otg.CurrentAcceleration[0] := 0;
otg.CurrentAcceleration[1] := 0.2;
otg.CurrentAcceleration[2] := 0;

otg.TargetPosition[0] := 1.0;
otg.TargetPosition[1] := -3.0;
otg.TargetPosition[2] := 2.0;

otg.TargetVelocity[0] := 0.0;
otg.TargetVelocity[1] := 0.0;
otg.TargetVelocity[2] := 0.2;

otg.TargetAcceleration[0] := 0.0;
otg.TargetAcceleration[1] := 0.0;
otg.TargetAcceleration[2] := -0.1;

otg.MaxVelocity[0] := 1;
otg.MaxVelocity[1] := 1;
otg.MaxVelocity[2] := 1;

otg.MaxAcceleration[0] := 1;
otg.MaxAcceleration[1] := 1;
otg.MaxAcceleration[2] := 1;

otg.MaxJerk[0] := 1;
otg.MaxJerk[1] := 1;
otg.MaxJerk[2] := 1;

otg(EnableAutoPropagate := FALSE);
result := otg.State;
AssertEquals_LREAL(otg.Duration, 3.6578610221, 1E-6, Message := ''); 

TEST_FINISHED();
END_METHOD

METHOD Test_FirstStateAtTime
VAR_INST
  otg : Struckig.Otg(0.005, 3) := (
  
    Synchronization := SynchronizationType.TimeSync,
    CurrentPosition :=     [ 0.0, -2.0, 0.0 ],
    CurrentVelocity :=     [ 0.0, 0.0, 0.0 ],
    CurrentAcceleration := [ 0.0, 0.0, 0.0 ],
    TargetPosition :=      [ 1.0, -3.0, 2.0 ],
    TargetVelocity :=      [ 0.0, 0.3, 0.0 ],
    TargetAcceleration :=  [ 0.0, 0.0, 0.0 ],
    MaxVelocity :=         [ 1.0, 1.0, 1.0 ],
    MaxAcceleration :=     [ 1.0, 1.0, 1.0 ],
    MaxJerk :=             [ 1.0, 1.0, 1.0 ]
  );
    
END_VAR
VAR
  result : Struckig.TrajectoryState;
  NewPosition, NewVelocity, NewAcceleration, values : ARRAY[0..Struckig.ParameterList.MaxDoFs] OF LREAL;
  positionExtrema : Struckig.PositionExtremaDesc;
  rtime, rvel, racc : LREAL;
END_VAR
TEST('FirstStateAtTime');

otg();

AssertTrue( otg._profiles[0].firstStateAtPosition(0.0, 0.0, rtime, rvel, racc), message:='' );
AssertEquals_LREAL(0.0, rtime, 1E-9, message:='');

AssertTrue( otg._profiles[0].firstStateAtPosition(0.5, 0.0, rtime, rvel, racc), message:='' );
AssertEquals_LREAL(2.0, rtime, 1E-9, message:='');

AssertTrue( otg._profiles[0].firstStateAtPosition(1.0, 0.0, rtime, rvel, racc), message:='' );
AssertEquals_LREAL(3.9999857615998957, rtime, 1E-9, message:=''); // doctest::Approx(4.0) 

AssertTrue( otg._profiles[1].firstStateAtPosition(-3.0, 0.0, rtime, rvel, racc), message:='' );
AssertEquals_LREAL(2.6004877902, rtime, 1E-9, message:='');

AssertTrue( otg._profiles[1].firstStateAtPosition(-3.1, 0.0, rtime, rvel, racc), message:='' );
AssertEquals_LREAL(2.8644154489, rtime, 1E-9, message:='');

AssertTrue( otg._profiles[2].firstStateAtPosition(0.05, 0.0, rtime, rvel, racc), message:='' );
AssertEquals_LREAL(0.6694329501, rtime, 1E-9, message:='');

AssertFalse( otg._profiles[0].firstStateAtPosition(-1.0, 0.0, rtime, rvel, racc), message:='' );
AssertFalse( otg._profiles[1].firstStateAtPosition(-3.4, 0.0, rtime, rvel, racc), message:='' );

// todo: this test doesn't make sense in the port of ruckig, the method is not exposed in the trajectory class yet
// AssertFalse( ruckig._profiles[6].firstStateAtPosition(6, 0.0, rtime, rvel, racc), message:='' );

TEST_FINISHED();
END_METHOD

METHOD Test_IndependentMinDurations
VAR_INST
  otg : Struckig.Otg(0.005, 3) := (
  
    Synchronization := SynchronizationType.None,
    CurrentPosition :=     [ 0.0, -2.0, 0.0 ],
    CurrentVelocity :=     [ 0.0, 0.0, 0.0 ],
    CurrentAcceleration := [ 0.0, 0.0, 0.0 ],
    TargetPosition :=      [ 1.0, -3.0, 2.0 ],
    TargetVelocity :=      [ 0.0, 0.3, 0.0 ],
    TargetAcceleration :=  [ 0.0, 0.0, 0.0 ],
    MaxVelocity :=         [ 1.0, 1.0, 1.0 ],
    MaxAcceleration :=     [ 1.0, 1.0, 1.0 ],
    MaxJerk :=             [ 1.0, 1.0, 1.0 ]
  );
    
END_VAR
VAR
  result : Struckig.TrajectoryState;
  NewPosition, NewVelocity, NewAcceleration, values : ARRAY[0..Struckig.ParameterList.MaxDoFs] OF LREAL;
  positionExtrema : Struckig.PositionExtremaDesc;
  rtime, rvel, racc : LREAL;
END_VAR
TEST('IndependentMinDurations');

otg();

AssertEquals_LREAL(otg._independentMinDurations[0], 3.1748021039, 1E-9, message:='');
AssertEquals_LREAL(otg._independentMinDurations[1], 3.6860977315, 1E-9, message:='');
AssertEquals_LREAL(otg._independentMinDurations[2], otg.Duration, 1E-9, message:='');

TEST_FINISHED();
END_METHOD

METHOD Test_InvalidInput
VAR_INST
  otg : Struckig.Otg(0.005, 3) := (
  
    Synchronization := SynchronizationType.None,
    CurrentPosition :=     [ 0.0, -2.0, 0.0 ],
    CurrentVelocity :=     [ 0.0, 0.0, 0.0 ],
    CurrentAcceleration := [ 0.0, 0.0, 0.0 ],
    TargetPosition :=      [ 1.0, -3.0, 2.0 ],
    TargetVelocity :=      [ 0.0, 0.3, 0.0 ],
    TargetAcceleration :=  [ 0.0, 0.0, 0.0 ],
    MaxVelocity :=         [ 1.0, 1.0, 1.0 ],
    MaxAcceleration :=     [ 1.0, 1.0, 1.0 ],
    MaxJerk :=             [ 1.0, 1.0, 1.0 ]
  );
    
END_VAR
VAR
  result : Struckig.TrajectoryState;
  NewPosition, NewVelocity, NewAcceleration, values : ARRAY[0..Struckig.ParameterList.MaxDoFs] OF LREAL;
  positionExtrema : Struckig.PositionExtremaDesc;
  rtime, rvel, racc : LREAL;
END_VAR
TEST('InvalidInput');

otg();

otg.TargetVelocity[0] := 2.0;
otg.TargetVelocity[1] := 0.3;
otg.TargetVelocity[2] := 0.0;

otg();

AssertEquals_INT(otg.State, Struckig.TrajectoryState.error, message:='State should be error');
AssertFalse(otg.NewCalculation, message:='ruckig.NewCalculation should be false');

otg.TargetVelocity[0] := 0.2;
otg.TargetVelocity[1] := -0.3;
otg.TargetVelocity[2] := 0.8;

otg();

AssertEquals_INT(otg.State, Struckig.TrajectoryState.busy, message:='State should be busy');
AssertTrue(otg.NewCalculation, message:='ruckig.NewCalculation should be true');

TEST_FINISHED();
END_METHOD

METHOD Test_PerDofSettings
VAR_INST
  otg : Struckig.Otg(0.005, 3) := (
    CurrentPosition :=     [ 0.0, -2.0, 0.0 ],
    CurrentVelocity :=     [ 0.0, 0.0, 0.0 ],
    CurrentAcceleration := [ 0.0, 0.0, 0.0 ],
    TargetPosition :=      [ 1.0, -3.0, 2.0 ],
    TargetVelocity :=      [ 0.0, 0.3, 0.0 ],
    TargetAcceleration :=  [ 0.0, 0.0, 0.0 ],
    MaxVelocity :=         [ 1.0, 1.0, 1.0 ],
    MaxAcceleration :=     [ 1.0, 1.0, 1.0 ],
    MaxJerk :=             [ 1.0, 1.0, 1.0 ]
  );
    
END_VAR
VAR
  result : Struckig.TrajectoryState;
  NewPosition, NewVelocity, NewAcceleration, values : ARRAY[0..Struckig.ParameterList.MaxDoFs] OF LREAL;
  NewSection : INT;
  positionExtrema : Struckig.PositionExtremaDesc;
  rtime, rvel, racc : LREAL;
END_VAR
TEST('PerDofSettings');

otg();
AssertEquals_INT(otg.State, Struckig.TrajectoryState.Busy, message:='State should be busy');
AssertEquals_LREAL(otg.Duration, 4, 1E-6, message:='Duration not met');

otg.AtTime(2.0, ADR(NewPosition), ADR(NewVelocity), ADR(NewAcceleration), ADR(NewSection));
values[0] := 0.5;
values[1] := -2.6871268303;
values[2] :=  1.0;
AssertArrayEquals_LREAL(values, NewPosition, 1E-6, message:='Position not met');


otg.ControlInterface := ControlInterfaceType.Velocity;
otg();
AssertEquals_INT(otg.State, Struckig.TrajectoryState.Busy, message:='State should be busy');
AssertEquals_LREAL(otg.Duration, 1.095445115, 1E-6, message:='Duration not met');

otg.AtTime(1.0, ADR(NewPosition), ADR(NewVelocity), ADR(NewAcceleration), ADR(NewSection));
values[0] := 0.0;
values[1] := -1.8641718534;
values[2] :=  0.0;
AssertArrayEquals_LREAL(values, NewPosition, 1E-6, message:='Position not met');


otg.PerDofControlInterface[0] := ControlInterfaceType.Position;
otg.PerDofControlInterface[1] := ControlInterfaceType.Velocity;
otg.PerDofControlInterface[2] := ControlInterfaceType.Position;
otg();
AssertEquals_INT(otg.State, Struckig.TrajectoryState.Busy, message:='State should be busy');
AssertEquals_LREAL(otg.Duration, 4.0, 1E-6, message:='Duration not met');

otg.AtTime(2.0, ADR(NewPosition), ADR(NewVelocity), ADR(NewAcceleration), ADR(NewSection));
values[0] := 0.5;
values[1] := -1.8528486838;
values[2] := 1.0;
AssertArrayEquals_LREAL(values, NewPosition, 1E-6, message:='Position not met');


otg.PerDofSynchronization[0] := SynchronizationType.TimeSync;
otg.PerDofSynchronization[1] := SynchronizationType.None;
otg.PerDofSynchronization[2] := SynchronizationType.TimeSync;
otg();
AssertEquals_INT(otg.State, Struckig.TrajectoryState.Busy, message:='State should be busy');
AssertEquals_LREAL(otg.Duration, 4.0, 1E-6, message:='Duration not met');

otg.AtTime(2.0, ADR(NewPosition), ADR(NewVelocity), ADR(NewAcceleration), ADR(NewSection));
values[0] := 0.5;
values[1] := -1.5643167673;
values[2] := 1.0;
AssertArrayEquals_LREAL(values, NewPosition, 1E-6, message:='Position not met');

otg.ControlInterface := ControlInterfaceType.Position;
otg.PerDofControlInterface[0] := ControlInterfaceType.Undefined;
otg.PerDofControlInterface[1] := ControlInterfaceType.Undefined;
otg.PerDofControlInterface[2] := ControlInterfaceType.Undefined;
otg.PerDofSynchronization[0] := SynchronizationType.None;
otg.PerDofSynchronization[1] := SynchronizationType.TimeSync;
otg.PerDofSynchronization[2] := SynchronizationType.TimeSync;
otg();
AssertEquals_INT(otg.State, Struckig.TrajectoryState.Busy, message:='State should be busy');
AssertEquals_LREAL(otg.Duration, 4.0, 1E-6, message:='Duration not met');

otg.AtTime(2.0, ADR(NewPosition), ADR(NewVelocity), ADR(NewAcceleration), ADR(NewSection));
values[0] := 0.7482143874;
values[1] := -2.6871268303;
values[2] := 1.0;
AssertArrayEquals_LREAL(values, NewPosition, 1E-6, message:='Position not met');

TEST_FINISHED();
END_METHOD

METHOD Test_PerDofSettings_1
VAR_INST
  otg : Struckig.Otg(0.005, 3) := (
    CurrentPosition :=     [ 0.0, 0.0, 0.0 ],
    CurrentVelocity :=     [ 0.0, 0.0, 0.0 ],
    CurrentAcceleration := [ 0.0, 0.0, 0.0 ],
    TargetPosition :=      [ 35, 35, 35 ],
    TargetVelocity :=      [ 125, 125, 100 ],
    TargetAcceleration :=  [ 0.0, 0.0, 0.0 ],
    MaxVelocity :=         [ 125, 125, 100 ],
    MaxAcceleration :=     [ 2000, 2000, 2000 ],
    MaxJerk :=             [ 20000, 20000, 20000 ]
  );
    
END_VAR
VAR
  result : Struckig.TrajectoryState;
END_VAR
TEST('PerDofSettings_1');

otg.ControlInterface := ControlInterfaceType.Position;
otg.PerDofControlInterface[0] := ControlInterfaceType.Undefined;
otg.PerDofControlInterface[1] := ControlInterfaceType.Undefined;
otg.PerDofControlInterface[2] := ControlInterfaceType.Undefined;
otg.PerDofSynchronization[0] := SynchronizationType.TimeSync;
otg.PerDofSynchronization[1] := SynchronizationType.TimeSync;
otg.PerDofSynchronization[2] := SynchronizationType.None;
otg();
AssertEquals_INT(otg.State, Struckig.TrajectoryState.Busy, message:='State should be busy');
AssertEquals_LREAL(otg.Duration, 0.4207106781, 1E-6, message:='Duration not met');


otg.CurrentPosition[0] := 0;
otg.CurrentPosition[1] := -2;
otg.CurrentPosition[2] := 0;

otg.CurrentVelocity[0] := 0;
otg.CurrentVelocity[1] := 0.2;
otg.CurrentVelocity[2] := 0;

otg.CurrentAcceleration[0] := 0;
otg.CurrentAcceleration[1] := 0.2;
otg.CurrentAcceleration[2] := 0;

otg.TargetPosition[0] := 1.0;
otg.TargetPosition[1] := -3.0;
otg.TargetPosition[2] := 2.0;

otg.TargetVelocity[0] := 0.0;
otg.TargetVelocity[1] := 0.0;
otg.TargetVelocity[2] := 0.2;

otg.TargetAcceleration[0] := 0.0;
otg.TargetAcceleration[1] := 0.0;
otg.TargetAcceleration[2] := -0.1;

otg.MaxVelocity[0] := 1;
otg.MaxVelocity[1] := 1;
otg.MaxVelocity[2] := 1;

otg.MaxAcceleration[0] := 1;
otg.MaxAcceleration[1] := 1;
otg.MaxAcceleration[2] := 1;

otg.MaxJerk[0] := 1;
otg.MaxJerk[1] := 1;
otg.MaxJerk[2] := 1;

otg.PerDofSynchronization[0] := SynchronizationType.None;
otg.PerDofSynchronization[1] := SynchronizationType.None;
otg.PerDofSynchronization[2] := SynchronizationType.TimeSync;

otg();
AssertEquals_INT(otg.State, Struckig.TrajectoryState.Busy, message:='State should be busy');
AssertEquals_LREAL(otg.Duration, 3.7885667284, 1E-6, message:='Duration not met');

otg.PerDofSynchronization[0] := SynchronizationType.None;
otg.PerDofSynchronization[1] := SynchronizationType.TimeSync;
otg.PerDofSynchronization[2] := SynchronizationType.None;

otg();
AssertEquals_INT(otg.State, Struckig.TrajectoryState.Busy, message:='State should be busy');
AssertEquals_LREAL(otg.Duration, 3.7885667284, 1E-6, message:='Duration not met');

otg.Enabled[0] := TRUE;
otg.Enabled[1] := FALSE;
otg.Enabled[2] := TRUE;

otg();
AssertEquals_INT(otg.State, Struckig.TrajectoryState.Busy, message:='State should be busy');
AssertEquals_LREAL(otg.Duration, 3.6578610221, 1E-6, message:='Duration not met');

TEST_FINISHED();
END_METHOD

METHOD Test_PhaseSynchronization
VAR_INST
  otg : Struckig.Otg(0.005, 3) := (
    Synchronization := SynchronizationType.Phase,
    CurrentPosition :=     [ 0.0, -2.0, 0.0 ],
    TargetPosition :=      [ 1.0, -3.0, 2.0 ],
    MaxVelocity :=         [ 1.0, 1.0, 1.0 ],
    MaxAcceleration :=     [ 1.0, 1.0, 1.0 ],
    MaxJerk :=             [ 1.0, 1.0, 1.0 ]
  ); 
END_VAR
VAR
  result : Struckig.TrajectoryState;
  busy : Struckig.TrajectoryState := Struckig.TrajectoryState.Busy;
  NewSection : INT;
  NewPosition, NewVelocity, NewAcceleration, values : ARRAY[0..Struckig.ParameterList.MaxDoFs] OF LREAL;
  positionExtrema : Struckig.PositionExtremaDesc;
  rtime, rvel, racc : LREAL;
END_VAR
TEST('PhaseSynchronization');

otg();
result := otg.State;
AssertEquals(busy, result, Message := '');
AssertEquals_LREAL(otg.Duration, 4.0, 1E-6, Message := ''); 
otg.AtTime(1.0, ADR(NewPosition), ADR(NewVelocity), ADR(NewAcceleration), ADR(NewSection));
values[0] := 0.0833333333;
values[1] := -2.0833333333;
values[2] := 0.1666666667;
AssertArrayEquals_LREAL(values, NewPosition, 1E-6, '');




otg.CurrentPosition[0] := 0.0;
otg.CurrentPosition[1] := -2.0;
otg.CurrentPosition[2] := 0.0;

otg.TargetPosition[0] := 10.0;
otg.TargetPosition[1] := -3.0;
otg.TargetPosition[2] := 2.0;

otg.MaxVelocity[0] := 10.0;
otg.MaxVelocity[1] := 2.0;
otg.MaxVelocity[2] := 1.0;

otg.MaxAcceleration[0] := 10.0;
otg.MaxAcceleration[1] := 2.0;
otg.MaxAcceleration[2] := 1.0;

otg.MaxJerk[0] := 10.0;
otg.MaxJerk[1] := 2.0;
otg.MaxJerk[2] := 1.0;

otg();
result := otg.State;
AssertEquals(busy, result, Message := '');
AssertEquals_LREAL(otg.Duration, 4.0, 1E-6, Message := ''); 
otg.AtTime(1.0, ADR(NewPosition), ADR(NewVelocity), ADR(NewAcceleration), ADR(NewSection));
values[0] := 0.8333333333;
values[1] := -2.0833333333;
values[2] := 0.1666666667;
AssertArrayEquals_LREAL(values, NewPosition, 1E-6, '');

TEST_FINISHED();
END_METHOD

METHOD Test_PositionExtrema
VAR_INST
  otg : Struckig.Otg(0.005, 3) := (
    Synchronization := SynchronizationType.TimeSync,
    CurrentPosition :=     [ 0.0, -2.0, 0.0 ],
    TargetPosition :=      [ 1.0, -3.0, 2.0 ],
    TargetVelocity :=      [ 0.0, 0.3, 0.0 ],
    MaxVelocity :=         [ 1.0, 1.0, 1.0 ],
    MaxAcceleration :=     [ 1.0, 1.0, 1.0 ],
    MaxJerk :=             [ 1.0, 1.0, 1.0 ]
  );     
END_VAR
VAR
  result : Struckig.TrajectoryState;
  NewPosition, NewVelocity, NewAcceleration, values : ARRAY[0..Struckig.ParameterList.MaxDoFs] OF LREAL;
  positionExtrema : Struckig.PositionExtremaDesc;
  rtime, rvel, racc : LREAL;
END_VAR
TEST('PositionExtrema');

otg();

positionExtrema := otg._profiles[0].positionExtrema();
AssertEquals_LREAL(4.0, positionExtrema.Tmax, 1E-9, message:='Profile[0] Tmax incorrect');
AssertEquals_LREAL(1.0, positionExtrema.Maximum, 1E-9, message:='Profile[0] maximum incorrect');
AssertEquals_LREAL(0.0, positionExtrema.Tmin, 1E-9, message:='Profile[0] Tmin incorrect');
AssertEquals_LREAL(0.0, positionExtrema.Minimum, 1E-9, message:='Profile[0] minimum incorrect');

positionExtrema := otg._profiles[1].positionExtrema();
AssertEquals_LREAL(0.0, positionExtrema.Tmax, 1E-9, message:='Profile[1] Tmax incorrect');
AssertEquals_LREAL(-2.0, positionExtrema.Maximum, 1E-9, message:='Profile[1] maximum incorrect');
AssertEquals_LREAL(3.2254033308, positionExtrema.Tmin, 1E-9, message:='Profile[1] Tmin incorrect');
AssertEquals_LREAL(-3.1549193338, positionExtrema.Minimum, 1E-9, message:='Profile[1] minimum incorrect');

positionExtrema := otg._profiles[2].positionExtrema();
AssertEquals_LREAL(4.0, positionExtrema.Tmax, 1E-9, message:='Profile[2] Tmax incorrect');
AssertEquals_LREAL(2.0, positionExtrema.Maximum, 1E-9, message:='Profile[2] maximum incorrect');
AssertEquals_LREAL(0.0, positionExtrema.Tmin, 1E-9, message:='Profile[2] Tmin incorrect');
AssertEquals_LREAL(0.0, positionExtrema.Minimum, 1E-9, message:='Profile[2] minimum incorrect');

TEST_FINISHED();
END_METHOD

END_FUNCTION_BLOCK

// ---- POUs/DebuggedExamplesTest.TcPOU
FUNCTION_BLOCK DebuggedExamplesTest EXTENDS TcUnit.FB_TestSuite

Test_Trajectory_HasTargetVelocity_HasTargetAcceleration();

METHOD Test_Trajectory_HasTargetVelocity_HasTargetAcceleration
VAR_INST
  ruckig : Struckig.Otg(0.001, 3) := (
  
    Synchronization := SynchronizationType.TimeSync,        
    MaxVelocity := [ 2000.00000000000000000000, 2000.00000000000000000000, 2000.00000000000000000000 ],
    MaxAcceleration := [ 20000.00000000000000000000, 20000.00000000000000000000, 20000.00000000000000000000 ],
    MaxJerk := [ 800000.00000000000000000000, 800000.00000000000000000000, 800000.00000000000000000000 ],
    CurrentPosition := [ -54.94342725690739825950, -71.16344937395382430623, -99.92141940871530891854 ],
    CurrentVelocity := [ 203.04708462957614756306, -87.88615914847480325989, -244.40742200449426491105 ],
    CurrentAcceleration := [ -9414.24830241836389177479, 3433.58972946014000626747, -1048.10905719350193976425 ],
    TargetPosition := [ -30.34627507739200780179, 41.33313071646210801191, 94.47974487226861128875 ],
    TargetVelocity := [ -104.33706621689987059654, -659.36109838358197521302, 811.33117925934993763804 ],
    TargetAcceleration := [ 523.43053514200096287823, 100.75104632855459385610, 320.80199262854853259341 ]
  );
  
  positionExtrema : Struckig.PositionExtremaDesc;
END_VAR
TEST('Trajectory_Profile[1]_Step2_TimeVel');

ruckig();

// Check total duration of profiles
AssertEquals_LREAL(Expected := 0.22338925049474450679, Actual := ruckig.Duration, DELTA := 1E-8, Message := 'Duration incorrect');

// Check duration for each phase
positionExtrema := ruckig._profiles[0].positionExtrema();
AssertEquals_LREAL(0.20657109030979783904, positionExtrema.Tmax, 1E-9, message:='Profile[0] Tmax incorrect');
AssertEquals_LREAL(-29.15176131633907630203, positionExtrema.Maximum, 1E-9, message:='Profile[0] maximum incorrect');
AssertEquals_LREAL(0.00000000000000000000, positionExtrema.Tmin, 1E-9, message:='Profile[0] Tmin incorrect');
AssertEquals_LREAL(-54.94342725690739825950, positionExtrema.Minimum, 1E-9, message:='Profile[0] minimum incorrect');

positionExtrema := ruckig._profiles[1].positionExtrema();
AssertEquals_LREAL(0.19826331168683380968, positionExtrema.Tmax, 1E-9, message:='Profile[1] Tmax incorrect');
AssertEquals_LREAL(55.81702313192161568622, positionExtrema.Maximum, 1E-9, message:='Profile[1] maximum incorrect');
AssertEquals_LREAL(0.01113968648909354625, positionExtrema.Tmin, 1E-9, message:='Profile[1] Tmin incorrect');
AssertEquals_LREAL(-71.74511835894615785492, positionExtrema.Minimum, 1E-9, message:='Profile[1] minimum incorrect');

positionExtrema := ruckig._profiles[2].positionExtrema();
AssertEquals_LREAL(0.22338925049474447904, positionExtrema.Tmax, 1E-9, message:='Profile[2] Tmax incorrect');
AssertEquals_LREAL(94.47974487226861128875, positionExtrema.Maximum, 1E-9, message:='Profile[2] maximum incorrect');
AssertEquals_LREAL(0.02606362117094545780, positionExtrema.Tmin, 1E-9, message:='Profile[2] Tmin incorrect');
AssertEquals_LREAL(-104.28684661857214166503, positionExtrema.Minimum, 1E-9, message:='Profile[2] minimum incorrect');
   

TEST_FINISHED();
END_METHOD

END_FUNCTION_BLOCK

// ---- POUs/TargetPosTest.TcPOU
FUNCTION_BLOCK TargetPosTest EXTENDS TcUnit.FB_TestSuite
VAR
  ruckig : Struckig.Otg(0.001, 3) := (
  
    Synchronization := SynchronizationType.TimeSync,        
    MaxVelocity := [ 2000.00000000000000000000, 2000.00000000000000000000, 2000.00000000000000000000 ],
    MaxAcceleration := [ 20000.00000000000000000000, 20000.00000000000000000000, 20000.00000000000000000000 ],
    MaxJerk := [ 800000.00000000000000000000, 800000.00000000000000000000, 800000.00000000000000000000 ],
    CurrentPosition := [ 48.86656216713086564596, 31.55963588984187140341, -13.09422790776093847853 ],
    CurrentVelocity := [ -274.21841080128081102885, -440.94461360926254656079, -764.75678162210920163488 ],
    CurrentAcceleration := [ -1478.09700836416959646158, 686.79611869591644790489, -9263.72976579731221136171 ],
    TargetPosition := [ 25.57994474955607699940, -15.83091418217283319336, -38.97164514571973370494 ],
    TargetVelocity := [ 0.00000000000000000000, 0.00000000000000000000, 0.00000000000000000000 ],
    TargetAcceleration := [ 0.00000000000000000000, 0.00000000000000000000, 0.00000000000000000000 ]
  );
  
  positionExtrema : Struckig.PositionExtremaDesc;  
END_VAR

Test_Trajectory_2();;
Test_Trajectory_5();
Test_Trajectory_6();
Test_Trajectory_7();
Test_Trajectory_12();
Test_Trajectory_16(); // this test required to do a more precise implementation of cbrt
Test_Trajectory_30();
Test_Trajectory_32();
Test_Trajectory_33();
Test_Trajectory_40();
Test_Trajectory_49();
Test_Trajectory_53();
Test_Trajectory_59();
Test_Trajectory_62();
Test_Trajectory_64();
Test_Trajectory_65();
Test_Trajectory_68();

METHOD Test_Trajectory_12
VAR_INST
  ruckig : Struckig.Otg(0.001, 3) := (
  
    Synchronization := SynchronizationType.TimeSync,        
    MaxVelocity := [ 2000.00000000000000000000, 2000.00000000000000000000, 2000.00000000000000000000 ],
    MaxAcceleration := [ 20000.00000000000000000000, 20000.00000000000000000000, 20000.00000000000000000000 ],
    MaxJerk := [ 800000.00000000000000000000, 800000.00000000000000000000, 800000.00000000000000000000 ],
    CurrentPosition := [ 12.15863849634686744139, 83.56438022017914590833, -29.82534868849941744884 ],
    CurrentVelocity := [ -881.54677264260010360886, -40.22247547933807254594, 795.30816871835008896596 ],
    CurrentAcceleration := [ 6802.73049394882036722265, -2844.95338607063877134351, -3652.21806306270900677191 ],
    TargetPosition := [ 61.24855302996508044089, -54.65891429617437324850, 65.64407005892678625969 ],
    TargetVelocity := [ 0.00000000000000000000, 0.00000000000000000000, 0.00000000000000000000 ],
    TargetAcceleration := [ 0.00000000000000000000, 0.00000000000000000000, 0.00000000000000000000 ]
  );
  
  positionExtrema : Struckig.PositionExtremaDesc;
END_VAR
TEST('Trajectory_12');

ruckig();

// Check total duration of profiles
AssertEquals_LREAL(Expected := 0.18765626933931714437, Actual := ruckig.Duration, DELTA := 1E-8, Message := 'Duration incorrect');

// Check duration for each phase
positionExtrema := ruckig._profiles[0].positionExtrema();
AssertEquals_LREAL(0.18765626933931711662, positionExtrema.Tmax, 1E-9, message:='Profile[0] Tmax incorrect');
AssertEquals_LREAL(61.24855302996508044089, positionExtrema.Maximum, 1E-9, message:='Profile[0] maximum incorrect');
AssertEquals_LREAL(0.01649658688256397387, positionExtrema.Tmin, 1E-9, message:='Profile[0] Tmin incorrect');
AssertEquals_LREAL(-0.85965741863935996037, positionExtrema.Minimum, 1E-9, message:='Profile[0] minimum incorrect');

positionExtrema := ruckig._profiles[1].positionExtrema();
AssertEquals_LREAL(0.00000000000000000000, positionExtrema.Tmax, 1E-9, message:='Profile[1] Tmax incorrect');
AssertEquals_LREAL(83.56438022017914590833, positionExtrema.Maximum, 1E-9, message:='Profile[1] maximum incorrect');
AssertEquals_LREAL(0.18765626933931714437, positionExtrema.Tmin, 1E-9, message:='Profile[1] Tmin incorrect');
AssertEquals_LREAL(-54.65891429617437324850, positionExtrema.Minimum, 1E-9, message:='Profile[1] minimum incorrect');

positionExtrema := ruckig._profiles[2].positionExtrema();
AssertEquals_LREAL(0.18765626933931711662, positionExtrema.Tmax, 1E-9, message:='Profile[2] Tmax incorrect');
AssertEquals_LREAL(65.64407005892678625969, positionExtrema.Maximum, 1E-9, message:='Profile[2] maximum incorrect');
AssertEquals_LREAL(0.00000000000000000000, positionExtrema.Tmin, 1E-9, message:='Profile[2] Tmin incorrect');
AssertEquals_LREAL(-29.82534868849941744884, positionExtrema.Minimum, 1E-9, message:='Profile[2] minimum incorrect');
   

TEST_FINISHED();
END_METHOD

METHOD Test_Trajectory_16
VAR_INST
  ruckig : Struckig.Otg(0.001, 3) := (
  
    Synchronization := SynchronizationType.TimeSync,        
    MaxVelocity := [ 2000.00000000000000000000, 2000.00000000000000000000, 2000.00000000000000000000 ],
    MaxAcceleration := [ 20000.00000000000000000000, 20000.00000000000000000000, 20000.00000000000000000000 ],
    MaxJerk := [ 800000.00000000000000000000, 800000.00000000000000000000, 800000.00000000000000000000 ],
    CurrentPosition := [ 8.21667911707363884943, -42.91905125747626215116, 48.44417367414695263506 ],
    CurrentVelocity := [ -786.82135287550590874162, 724.24582523622666485608, -678.96507198447488917736 ],
    CurrentAcceleration := [ 2775.55640569175011478364, 5006.65330127050037845038, -1991.17849814757664717035 ],
    TargetPosition := [ -91.18523630560480341956, 39.65724384459844031880, 80.00859285567460688071 ],
    TargetVelocity := [ 0.00000000000000000000, 0.00000000000000000000, 0.00000000000000000000 ],
    TargetAcceleration := [ 0.00000000000000000000, 0.00000000000000000000, 0.00000000000000000000 ]
  );
  
  positionExtrema : Struckig.PositionExtremaDesc;
END_VAR
TEST('Trajectory_16');

ruckig();

// Check total duration of profiles
AssertEquals_LREAL(Expected := 0.16787256653000462436, Actual := ruckig.Duration, DELTA := 1E-8, Message := 'Duration incorrect');

// Check duration for each phase
positionExtrema := ruckig._profiles[0].positionExtrema();
AssertEquals_LREAL(0, positionExtrema.Tmax, 1E-9, message:='Profile[0] Tmax incorrect');
AssertEquals_LREAL(8.2166791170736388494, positionExtrema.Maximum, 1E-9, message:='Profile[0] maximum incorrect');
AssertEquals_LREAL(0.16787256653000462436, positionExtrema.Tmin, 1E-9, message:='Profile[0] Tmin incorrect');
AssertEquals_LREAL(-91.18523630560480342, positionExtrema.Minimum, 1E-9, message:='Profile[0] minimum incorrect');

positionExtrema := ruckig._profiles[1].positionExtrema();
AssertEquals_LREAL(0.16787256609842091115, positionExtrema.Tmax, 1E-9, message:='Profile[1] Tmax incorrect');
AssertEquals_LREAL(39.657243844598482951, positionExtrema.Maximum, 1E-9, message:='Profile[1] maximum incorrect');
AssertEquals_LREAL(0, positionExtrema.Tmin, 1E-9, message:='Profile[1] Tmin incorrect');
AssertEquals_LREAL(-42.919051257476262151, positionExtrema.Minimum, 1E-9, message:='Profile[1] minimum incorrect');

positionExtrema := ruckig._profiles[2].positionExtrema();
AssertEquals_LREAL(0.16787256609842091115, positionExtrema.Tmax, 1E-9, message:='Profile[2] Tmax incorrect');
AssertEquals_LREAL(80.008592855674606881, positionExtrema.Maximum, 1E-9, message:='Profile[2] maximum incorrect');
AssertEquals_LREAL(0.027488973122684470102, positionExtrema.Tmin, 1E-9, message:='Profile[2] Tmin incorrect');
AssertEquals_LREAL(31.797392745296477301, positionExtrema.Minimum, 1E-9, message:='Profile[2] minimum incorrect');
   

TEST_FINISHED();
END_METHOD

METHOD Test_Trajectory_2
VAR_INST
  ruckig : Struckig.Otg(0.001, 3) := (
  
    Synchronization := SynchronizationType.TimeSync,        
    MaxVelocity := [ 2000.00000000000000000000, 2000.00000000000000000000, 2000.00000000000000000000 ],
    MaxAcceleration := [ 20000.00000000000000000000, 20000.00000000000000000000, 20000.00000000000000000000 ],
    MaxJerk := [ 800000.00000000000000000000, 800000.00000000000000000000, 800000.00000000000000000000 ],
    CurrentPosition := [ 44.74559775494429914033, 63.66880079927278757168, -12.48356919175202506267 ],
    CurrentVelocity := [ 264.84303106023071450181, -712.27423462239960372244, -643.21373646696986270399 ],
    CurrentAcceleration := [ 424.20358939641846518498, -6495.14198884339384676423, -9831.31287541736855928320 ],
    TargetPosition := [ 57.39429753248339238780, 42.08707495871314563374, -1.97763153852878303951 ],
    TargetVelocity := [ 0.00000000000000000000, 0.00000000000000000000, 0.00000000000000000000 ],
    TargetAcceleration := [ 0.00000000000000000000, 0.00000000000000000000, 0.00000000000000000000 ]
  );
  
  positionExtrema : Struckig.PositionExtremaDesc;
END_VAR
TEST('Trajectory_2');

ruckig();

// Check total duration of profiles
AssertEquals_LREAL(Expected := 0.16542491911229942336, Actual := ruckig.Duration, DELTA := 1E-8, Message := 'Duration incorrect');

// Check duration for each phase
positionExtrema := ruckig._profiles[0].positionExtrema();
AssertEquals_LREAL(0.16542491892541816290, positionExtrema.Tmax, 1E-9, message:='Profile[0] Tmax incorrect');
AssertEquals_LREAL(57.39429753248339949323, positionExtrema.Maximum, 1E-9, message:='Profile[0] maximum incorrect');
AssertEquals_LREAL(0.00000000000000000000, positionExtrema.Tmin, 1E-9, message:='Profile[0] Tmin incorrect');
AssertEquals_LREAL(44.74559775494429914033, positionExtrema.Minimum, 1E-9, message:='Profile[0] minimum incorrect');

positionExtrema := ruckig._profiles[1].positionExtrema();
AssertEquals_LREAL(0.00000000000000000000, positionExtrema.Tmax, 1E-9, message:='Profile[1] Tmax incorrect');
AssertEquals_LREAL(63.66880079927278757168, positionExtrema.Maximum, 1E-9, message:='Profile[1] maximum incorrect');
AssertEquals_LREAL(0.06011117382266835396, positionExtrema.Tmin, 1E-9, message:='Profile[1] Tmin incorrect');
AssertEquals_LREAL(35.26367745920458673936, positionExtrema.Minimum, 1E-9, message:='Profile[1] minimum incorrect');

positionExtrema := ruckig._profiles[2].positionExtrema();
AssertEquals_LREAL(0.16542491911229942336, positionExtrema.Tmax, 1E-9, message:='Profile[2] Tmax incorrect');
AssertEquals_LREAL(-1.97763153852878303951, positionExtrema.Maximum, 1E-9, message:='Profile[2] maximum incorrect');
AssertEquals_LREAL(0.08144760340330899073, positionExtrema.Tmin, 1E-9, message:='Profile[2] Tmin incorrect');
AssertEquals_LREAL(-36.92186481482234938767, positionExtrema.Minimum, 1E-9, message:='Profile[2] minimum incorrect');
   

TEST_FINISHED();
END_METHOD

METHOD Test_Trajectory_30
VAR_INST
  ruckig : Struckig.Otg(0.001, 3) := (
  
    Synchronization := SynchronizationType.TimeSync,        
    MaxVelocity := [ 2000.00000000000000000000, 2000.00000000000000000000, 2000.00000000000000000000 ],
    MaxAcceleration := [ 20000.00000000000000000000, 20000.00000000000000000000, 20000.00000000000000000000 ],
    MaxJerk := [ 800000.00000000000000000000, 800000.00000000000000000000, 800000.00000000000000000000 ],
    CurrentPosition := [ 20.18249544120934046987, -10.33662927823941402039, -59.33613032688207766796 ],
    CurrentVelocity := [ -147.36941969263784812938, 276.37127321170169125253, -471.16528659637026521523 ],
    CurrentAcceleration := [ 5958.91709773212642176077, -6024.30381588076943444321, 4027.41742253926349803805 ],
    TargetPosition := [ 57.35278694063060811459, 37.88908861774962133495, 47.84009680376084361342 ],
    TargetVelocity := [ 0.00000000000000000000, 0.00000000000000000000, 0.00000000000000000000 ],
    TargetAcceleration := [ 0.00000000000000000000, 0.00000000000000000000, 0.00000000000000000000 ]
  );
  
  positionExtrema : Struckig.PositionExtremaDesc;
END_VAR
TEST('Trajectory_30');

ruckig();

// Check total duration of profiles
AssertEquals_LREAL(Expected := 0.19875826019833076064, Actual := ruckig.Duration, DELTA := 1E-8, Message := 'Duration incorrect');

// Check duration for each phase
positionExtrema := ruckig._profiles[0].positionExtrema();
AssertEquals_LREAL(0.19875826019833078839, positionExtrema.Tmax, 1E-9, message:='Profile[0] Tmax incorrect');
AssertEquals_LREAL(57.35278694063060811459, positionExtrema.Maximum, 1E-9, message:='Profile[0] maximum incorrect');
AssertEquals_LREAL(0.01314032839612196309, positionExtrema.Tmin, 1E-9, message:='Profile[0] Tmin incorrect');
AssertEquals_LREAL(19.06299300602372071012, positionExtrema.Minimum, 1E-9, message:='Profile[0] minimum incorrect');

positionExtrema := ruckig._profiles[1].positionExtrema();
AssertEquals_LREAL(0.19875826019833076064, positionExtrema.Tmax, 1E-9, message:='Profile[1] Tmax incorrect');
AssertEquals_LREAL(37.88908861774962133495, positionExtrema.Maximum, 1E-9, message:='Profile[1] maximum incorrect');
AssertEquals_LREAL(0.00000000000000000000, positionExtrema.Tmin, 1E-9, message:='Profile[1] Tmin incorrect');
AssertEquals_LREAL(-10.33662927823941402039, positionExtrema.Minimum, 1E-9, message:='Profile[1] minimum incorrect');

positionExtrema := ruckig._profiles[2].positionExtrema();
AssertEquals_LREAL(0.19875826019833076064, positionExtrema.Tmax, 1E-9, message:='Profile[2] Tmax incorrect');
AssertEquals_LREAL(47.84009680376084361342, positionExtrema.Maximum, 1E-9, message:='Profile[2] maximum incorrect');
AssertEquals_LREAL(0.01996572822182592077, positionExtrema.Tmin, 1E-9, message:='Profile[2] Tmin incorrect');
AssertEquals_LREAL(-66.87937049880544293501, positionExtrema.Minimum, 1E-9, message:='Profile[2] minimum incorrect');
   

TEST_FINISHED();
END_METHOD

METHOD Test_Trajectory_32
VAR_INST
  ruckig : Struckig.Otg(0.001, 3) := (
  
    Synchronization := SynchronizationType.TimeSync,        
    MaxVelocity := [ 2000.00000000000000000000, 2000.00000000000000000000, 2000.00000000000000000000 ],
    MaxAcceleration := [ 20000.00000000000000000000, 20000.00000000000000000000, 20000.00000000000000000000 ],
    MaxJerk := [ 800000.00000000000000000000, 800000.00000000000000000000, 800000.00000000000000000000 ],
    CurrentPosition := [ -71.32072487430589546875, 75.77874394332496876814, -31.17619673281745917848 ],
    CurrentVelocity := [ -39.37043543026334191381, -314.80982911633589083067, -743.63983854388607142027 ],
    CurrentAcceleration := [ 918.61171848468075040728, -8240.24070744882010330912, 376.40421615367449703626 ],
    TargetPosition := [ -38.32577323859909057546, 76.88839801585137934126, 77.24450399202348194194 ],
    TargetVelocity := [ 0.00000000000000000000, 0.00000000000000000000, 0.00000000000000000000 ],
    TargetAcceleration := [ 0.00000000000000000000, 0.00000000000000000000, 0.00000000000000000000 ]
  );
  
  positionExtrema : Struckig.PositionExtremaDesc;
END_VAR
TEST('Trajectory_32');

ruckig();

// Check total duration of profiles
AssertEquals_LREAL(Expected := 0.22561874467077386308, Actual := ruckig.Duration, DELTA := 1E-8, Message := 'Duration incorrect');

// Check duration for each phase
positionExtrema := ruckig._profiles[0].positionExtrema();
AssertEquals_LREAL(0.22561874467077389084, positionExtrema.Tmax, 1E-9, message:='Profile[0] Tmax incorrect');
AssertEquals_LREAL(-38.32577323859909057546, positionExtrema.Maximum, 1E-9, message:='Profile[0] maximum incorrect');
AssertEquals_LREAL(0.00883895720172546244, positionExtrema.Tmin, 1E-9, message:='Profile[0] Tmin incorrect');
AssertEquals_LREAL(-71.54075918203305661791, positionExtrema.Minimum, 1E-9, message:='Profile[0] minimum incorrect');

positionExtrema := ruckig._profiles[1].positionExtrema();
AssertEquals_LREAL(0.22561874448389260261, positionExtrema.Tmax, 1E-9, message:='Profile[1] Tmax incorrect');
AssertEquals_LREAL(76.88839801585137934126, positionExtrema.Maximum, 1E-9, message:='Profile[1] maximum incorrect');
AssertEquals_LREAL(0.04326693976782886031, positionExtrema.Tmin, 1E-9, message:='Profile[1] Tmin incorrect');
AssertEquals_LREAL(64.99037106700389188063, positionExtrema.Minimum, 1E-9, message:='Profile[1] minimum incorrect');

positionExtrema := ruckig._profiles[2].positionExtrema();
AssertEquals_LREAL(0.22561874467077386308, positionExtrema.Tmax, 1E-9, message:='Profile[2] Tmax incorrect');
AssertEquals_LREAL(77.24450399202348194194, positionExtrema.Maximum, 1E-9, message:='Profile[2] maximum incorrect');
AssertEquals_LREAL(0.02452949472980790746, positionExtrema.Tmin, 1E-9, message:='Profile[2] Tmin incorrect');
AssertEquals_LREAL(-47.33615887649365561174, positionExtrema.Minimum, 1E-9, message:='Profile[2] minimum incorrect');
   

TEST_FINISHED();
END_METHOD

METHOD Test_Trajectory_33
VAR_INST
  ruckig : Struckig.Otg(0.001, 3) := (
  
    Synchronization := SynchronizationType.TimeSync,        
    MaxVelocity := [ 2000.00000000000000000000, 2000.00000000000000000000, 2000.00000000000000000000 ],
    MaxAcceleration := [ 20000.00000000000000000000, 20000.00000000000000000000, 20000.00000000000000000000 ],
    MaxJerk := [ 800000.00000000000000000000, 800000.00000000000000000000, 800000.00000000000000000000 ],
    CurrentPosition := [ -10.72081173000827902797, -58.44147038088563306246, 98.86324493851924444243 ],
    CurrentVelocity := [ -408.47451658779903027607, -786.19958599415508615493, -998.10812621012325962511 ],
    CurrentAcceleration := [ 3503.92425371204808470793, 3035.68280271572984929662, -8529.36175578239635797217 ],
    TargetPosition := [ -24.74505052699171869790, -29.66847304289291287205, -86.07591857423138037575 ],
    TargetVelocity := [ 0.00000000000000000000, 0.00000000000000000000, 0.00000000000000000000 ],
    TargetAcceleration := [ 0.00000000000000000000, 0.00000000000000000000, 0.00000000000000000000 ]
  );
  
  positionExtrema : Struckig.PositionExtremaDesc;
END_VAR
TEST('Trajectory_33');

ruckig();

// Check total duration of profiles
AssertEquals_LREAL(Expected := 0.17123630970102474147, Actual := ruckig.Duration, DELTA := 1E-8, Message := 'Duration incorrect');

// Check duration for each phase
positionExtrema := ruckig._profiles[0].positionExtrema();
AssertEquals_LREAL(0.00000000000000000000, positionExtrema.Tmax, 1E-9, message:='Profile[0] Tmax incorrect');
AssertEquals_LREAL(-10.72081173000827902797, positionExtrema.Maximum, 1E-9, message:='Profile[0] maximum incorrect');
AssertEquals_LREAL(0.17123630970102476923, positionExtrema.Tmin, 1E-9, message:='Profile[0] Tmin incorrect');
AssertEquals_LREAL(-24.74505052699171869790, positionExtrema.Minimum, 1E-9, message:='Profile[0] minimum incorrect');

positionExtrema := ruckig._profiles[1].positionExtrema();
AssertEquals_LREAL(0.17123630970102471371, positionExtrema.Tmax, 1E-9, message:='Profile[1] Tmax incorrect');
AssertEquals_LREAL(-29.66847304289291287205, positionExtrema.Maximum, 1E-9, message:='Profile[1] maximum incorrect');
AssertEquals_LREAL(0.06908515615955748701, positionExtrema.Tmin, 1E-9, message:='Profile[1] Tmin incorrect');
AssertEquals_LREAL(-76.18339289032344652242, positionExtrema.Minimum, 1E-9, message:='Profile[1] minimum incorrect');

positionExtrema := ruckig._profiles[2].positionExtrema();
AssertEquals_LREAL(0.00000000000000000000, positionExtrema.Tmax, 1E-9, message:='Profile[2] Tmax incorrect');
AssertEquals_LREAL(98.86324493851924444243, positionExtrema.Maximum, 1E-9, message:='Profile[2] maximum incorrect');
AssertEquals_LREAL(0.17123630970102474147, positionExtrema.Tmin, 1E-9, message:='Profile[2] Tmin incorrect');
AssertEquals_LREAL(-86.07591857423138037575, positionExtrema.Minimum, 1E-9, message:='Profile[2] minimum incorrect');
   

TEST_FINISHED();
END_METHOD

METHOD Test_Trajectory_40
VAR_INST
  ruckig : Struckig.Otg(0.001, 3) := (
  
    Synchronization := SynchronizationType.TimeSync,        
    MaxVelocity := [ 2000.00000000000000000000, 2000.00000000000000000000, 2000.00000000000000000000 ],
    MaxAcceleration := [ 20000.00000000000000000000, 20000.00000000000000000000, 20000.00000000000000000000 ],
    MaxJerk := [ 800000.00000000000000000000, 800000.00000000000000000000, 800000.00000000000000000000 ],
    CurrentPosition := [ 29.38520952151498022431, 0.54024576846694571941, -55.20826603737940274641 ],
    CurrentVelocity := [ -969.77050425776712927473, -274.95655325444397476531, 136.62875181670483470953 ],
    CurrentAcceleration := [ -3024.14261213553436391521, 816.78995976388432609383, -4328.68204209528175852029 ],
    TargetPosition := [ 1.97730433317153142525, -41.44239712071811254646, -63.08579022434781791162 ],
    TargetVelocity := [ 0.00000000000000000000, 0.00000000000000000000, 0.00000000000000000000 ],
    TargetAcceleration := [ 0.00000000000000000000, 0.00000000000000000000, 0.00000000000000000000 ]
  );
  
  positionExtrema : Struckig.PositionExtremaDesc;
END_VAR
TEST('Trajectory_40');

ruckig();

// Check total duration of profiles
AssertEquals_LREAL(Expected := 0.13217815288228063064, Actual := ruckig.Duration, DELTA := 1E-8, Message := 'Duration incorrect');

// Check duration for each phase
positionExtrema := ruckig._profiles[0].positionExtrema();
AssertEquals_LREAL(0.00000000000000000000, positionExtrema.Tmax, 1E-9, message:='Profile[0] Tmax incorrect');
AssertEquals_LREAL(29.38520952151498022431, positionExtrema.Maximum, 1E-9, message:='Profile[0] maximum incorrect');
AssertEquals_LREAL(0.06794606535212494025, positionExtrema.Tmin, 1E-9, message:='Profile[0] Tmin incorrect');
AssertEquals_LREAL(-9.67357879957821609196, positionExtrema.Minimum, 1E-9, message:='Profile[0] minimum incorrect');

positionExtrema := ruckig._profiles[1].positionExtrema();
AssertEquals_LREAL(0.00000000000000000000, positionExtrema.Tmax, 1E-9, message:='Profile[1] Tmax incorrect');
AssertEquals_LREAL(0.54024576846694571941, positionExtrema.Maximum, 1E-9, message:='Profile[1] maximum incorrect');
AssertEquals_LREAL(0.13217815288228063064, positionExtrema.Tmin, 1E-9, message:='Profile[1] Tmin incorrect');
AssertEquals_LREAL(-41.44239712071811254646, positionExtrema.Minimum, 1E-9, message:='Profile[1] minimum incorrect');

positionExtrema := ruckig._profiles[2].positionExtrema();
AssertEquals_LREAL(0.01413581147570610458, positionExtrema.Tmax, 1E-9, message:='Profile[2] Tmax incorrect');
AssertEquals_LREAL(-54.08246211603182018735, positionExtrema.Maximum, 1E-9, message:='Profile[2] maximum incorrect');
AssertEquals_LREAL(0.13217815261799065185, positionExtrema.Tmin, 1E-9, message:='Profile[2] Tmin incorrect');
AssertEquals_LREAL(-63.08579022434781791162, positionExtrema.Minimum, 1E-9, message:='Profile[2] minimum incorrect');
   

TEST_FINISHED();
END_METHOD

METHOD Test_Trajectory_49
VAR_INST
  ruckig : Struckig.Otg(0.001, 3) := (
  
    Synchronization := SynchronizationType.TimeSync,        
    MaxVelocity := [ 2000.00000000000000000000, 2000.00000000000000000000, 2000.00000000000000000000 ],
    MaxAcceleration := [ 20000.00000000000000000000, 20000.00000000000000000000, 20000.00000000000000000000 ],
    MaxJerk := [ 800000.00000000000000000000, 800000.00000000000000000000, 800000.00000000000000000000 ],
    CurrentPosition := [ -29.51211691133248393726, -68.13722912354262462031, 25.86635819923048984492 ],
    CurrentVelocity := [ -361.39127939828188118554, 280.60480492296255761175, 432.98890733596567770292 ],
    CurrentAcceleration := [ -4470.60901176135485002305, 6427.77132791660551447421, -7455.37531375192429550225 ],
    TargetPosition := [ 60.41587137499075765845, -7.73628974565106375394, 93.39422462833789495562 ],
    TargetVelocity := [ 0.00000000000000000000, 0.00000000000000000000, 0.00000000000000000000 ],
    TargetAcceleration := [ 0.00000000000000000000, 0.00000000000000000000, 0.00000000000000000000 ]
  );
  
  positionExtrema : Struckig.PositionExtremaDesc;
END_VAR
TEST('Trajectory_49');

ruckig();

// Check total duration of profiles
AssertEquals_LREAL(Expected := 0.19300944274036524462, Actual := ruckig.Duration, DELTA := 1E-8, Message := 'Duration incorrect');

// Check duration for each phase
positionExtrema := ruckig._profiles[0].positionExtrema();
AssertEquals_LREAL(0.19300944274036524462, positionExtrema.Tmax, 1E-9, message:='Profile[0] Tmax incorrect');
AssertEquals_LREAL(60.41587137499075765845, positionExtrema.Maximum, 1E-9, message:='Profile[0] maximum incorrect');
AssertEquals_LREAL(0.03058826126470169660, positionExtrema.Tmin, 1E-9, message:='Profile[0] Tmin incorrect');
AssertEquals_LREAL(-38.84193813948969165040, positionExtrema.Minimum, 1E-9, message:='Profile[0] minimum incorrect');

positionExtrema := ruckig._profiles[1].positionExtrema();
AssertEquals_LREAL(0.19300944274036524462, positionExtrema.Tmax, 1E-9, message:='Profile[1] Tmax incorrect');
AssertEquals_LREAL(-7.73628974565106375394, positionExtrema.Maximum, 1E-9, message:='Profile[1] maximum incorrect');
AssertEquals_LREAL(0.00000000000000000000, positionExtrema.Tmin, 1E-9, message:='Profile[1] Tmin incorrect');
AssertEquals_LREAL(-68.13722912354262462031, positionExtrema.Minimum, 1E-9, message:='Profile[1] minimum incorrect');

positionExtrema := ruckig._profiles[2].positionExtrema();
AssertEquals_LREAL(0.19300944274036524462, positionExtrema.Tmax, 1E-9, message:='Profile[2] Tmax incorrect');
AssertEquals_LREAL(93.39422462833789495562, positionExtrema.Maximum, 1E-9, message:='Profile[2] maximum incorrect');
AssertEquals_LREAL(0.00000000000000000000, positionExtrema.Tmin, 1E-9, message:='Profile[2] Tmin incorrect');
AssertEquals_LREAL(25.86635819923048984492, positionExtrema.Minimum, 1E-9, message:='Profile[2] minimum incorrect');
   

TEST_FINISHED();
END_METHOD

METHOD Test_Trajectory_5
VAR_INST
  ruckig : Struckig.Otg(0.001, 3) := (
  
    Synchronization := SynchronizationType.TimeSync,        
    MaxVelocity := [ 2000.00000000000000000000, 2000.00000000000000000000, 2000.00000000000000000000 ],
    MaxAcceleration := [ 20000.00000000000000000000, 20000.00000000000000000000, 20000.00000000000000000000 ],
    MaxJerk := [ 800000.00000000000000000000, 800000.00000000000000000000, 800000.00000000000000000000 ],
    CurrentPosition := [ -56.80336446239233794131, -86.51356035578187686497, -74.10635479722176910400 ],
    CurrentVelocity := [ -592.89949250113568268716, -990.58767738485028075957, 657.50930880589612570475 ],
    CurrentAcceleration := [ 1441.54985938923709909432, 5942.57310535894430358894, 9734.30059765397891169414 ],
    TargetPosition := [ -19.92529957498598491838, -6.87084002731369025696, 65.89578231878417113876 ],
    TargetVelocity := [ 0.00000000000000000000, 0.00000000000000000000, 0.00000000000000000000 ],
    TargetAcceleration := [ 0.00000000000000000000, 0.00000000000000000000, 0.00000000000000000000 ]
  );
  
  positionExtrema : Struckig.PositionExtremaDesc;
END_VAR
TEST('Trajectory_5');

ruckig();

// Check total duration of profiles
AssertEquals_LREAL(Expected := 0.21893317752843077795, Actual := ruckig.Duration, DELTA := 1E-8, Message := 'Duration incorrect');

// Check duration for each phase
positionExtrema := ruckig._profiles[0].positionExtrema();
AssertEquals_LREAL(0.21893317722325497665, positionExtrema.Tmax, 1E-9, message:='Profile[0] Tmax incorrect');
AssertEquals_LREAL(-19.92529957498598491838, positionExtrema.Maximum, 1E-9, message:='Profile[0] maximum incorrect');
AssertEquals_LREAL(0.04539326985447761365, positionExtrema.Tmin, 1E-9, message:='Profile[0] Tmin incorrect');
AssertEquals_LREAL(-71.21834027209614248477, positionExtrema.Minimum, 1E-9, message:='Profile[0] minimum incorrect');

positionExtrema := ruckig._profiles[1].positionExtrema();
AssertEquals_LREAL(0.21893317699985082037, positionExtrema.Tmax, 1E-9, message:='Profile[1] Tmax incorrect');
AssertEquals_LREAL(-6.87084002731364940075, positionExtrema.Maximum, 1E-9, message:='Profile[1] maximum incorrect');
AssertEquals_LREAL(0.01757178361830132041, positionExtrema.Tmin, 1E-9, message:='Profile[1] Tmin incorrect');
AssertEquals_LREAL(-102.27910277467870514556, positionExtrema.Minimum, 1E-9, message:='Profile[1] minimum incorrect');

positionExtrema := ruckig._profiles[2].positionExtrema();
AssertEquals_LREAL(0.21893317752843075019, positionExtrema.Tmax, 1E-9, message:='Profile[2] Tmax incorrect');
AssertEquals_LREAL(65.89578231878417113876, positionExtrema.Maximum, 1E-9, message:='Profile[2] maximum incorrect');
AssertEquals_LREAL(0.00000000000000000000, positionExtrema.Tmin, 1E-9, message:='Profile[2] Tmin incorrect');
AssertEquals_LREAL(-74.10635479722176910400, positionExtrema.Minimum, 1E-9, message:='Profile[2] minimum incorrect');
   

TEST_FINISHED();
END_METHOD

METHOD Test_Trajectory_53
VAR_INST
  ruckig : Struckig.Otg(0.001, 3) := (
  
    Synchronization := SynchronizationType.TimeSync,        
    MaxVelocity := [ 2000.00000000000000000000, 2000.00000000000000000000, 2000.00000000000000000000 ],
    MaxAcceleration := [ 20000.00000000000000000000, 20000.00000000000000000000, 20000.00000000000000000000 ],
    MaxJerk := [ 800000.00000000000000000000, 800000.00000000000000000000, 800000.00000000000000000000 ],
    CurrentPosition := [ 49.63749459770096450484, -62.67069199879444596490, 94.53868838473144364798 ],
    CurrentVelocity := [ 664.16399550988307964872, 189.17863757101872579369, -166.93673264110304899077 ],
    CurrentAcceleration := [ 3813.89534506026757298969, -4230.27473187632494955324, -810.58367009230460098479 ],
    TargetPosition := [ 40.02418382022895571026, 1.64383018244964773658, -62.79757540961892203768 ],
    TargetVelocity := [ 0.00000000000000000000, 0.00000000000000000000, 0.00000000000000000000 ],
    TargetAcceleration := [ 0.00000000000000000000, 0.00000000000000000000, 0.00000000000000000000 ]
  );
  
  positionExtrema : Struckig.PositionExtremaDesc;
END_VAR
TEST('Trajectory_53');

ruckig();

// Check total duration of profiles
AssertEquals_LREAL(Expected := 0.19412157092543416703, Actual := ruckig.Duration, DELTA := 1E-8, Message := 'Duration incorrect');

// Check duration for each phase
positionExtrema := ruckig._profiles[0].positionExtrema();
AssertEquals_LREAL(0.05226266454630152519, positionExtrema.Tmax, 1E-9, message:='Profile[0] Tmax incorrect');
AssertEquals_LREAL(72.04161381570744993041, positionExtrema.Maximum, 1E-9, message:='Profile[0] maximum incorrect');
AssertEquals_LREAL(0.19412157039685418169, positionExtrema.Tmin, 1E-9, message:='Profile[0] Tmin incorrect');
AssertEquals_LREAL(40.02418382022894860484, positionExtrema.Minimum, 1E-9, message:='Profile[0] minimum incorrect');

positionExtrema := ruckig._profiles[1].positionExtrema();
AssertEquals_LREAL(0.19412157092543416703, positionExtrema.Tmax, 1E-9, message:='Profile[1] Tmax incorrect');
AssertEquals_LREAL(1.64383018244964773658, positionExtrema.Maximum, 1E-9, message:='Profile[1] maximum incorrect');
AssertEquals_LREAL(0.00000000000000000000, positionExtrema.Tmin, 1E-9, message:='Profile[1] Tmin incorrect');
AssertEquals_LREAL(-62.67069199879444596490, positionExtrema.Minimum, 1E-9, message:='Profile[1] minimum incorrect');

positionExtrema := ruckig._profiles[2].positionExtrema();
AssertEquals_LREAL(0.00000000000000000000, positionExtrema.Tmax, 1E-9, message:='Profile[2] Tmax incorrect');
AssertEquals_LREAL(94.53868838473144364798, positionExtrema.Maximum, 1E-9, message:='Profile[2] maximum incorrect');
AssertEquals_LREAL(0.19412157092543416703, positionExtrema.Tmin, 1E-9, message:='Profile[2] Tmin incorrect');
AssertEquals_LREAL(-62.79757540961892203768, positionExtrema.Minimum, 1E-9, message:='Profile[2] minimum incorrect');
   

TEST_FINISHED();
END_METHOD

METHOD Test_Trajectory_59
VAR_INST

END_VAR
TEST('Trajectory_59');

ruckig();

// Check total duration of profiles
AssertEquals_LREAL(Expected := 0.12819874947134405, Actual := ruckig.Duration, DELTA := 1E-8, Message := 'Duration incorrect');
// this test returns the same values as the ruckig cpp version it is compiled with,
// but the newest version results differ

// Check duration for each phase
positionExtrema := ruckig._profiles[0].positionExtrema();
AssertEquals_LREAL(0.00000000000000000000, positionExtrema.Tmax, 1E-9, message:='Profile[0] Tmax incorrect');
AssertEquals_LREAL(48.86656216713086564596, positionExtrema.Maximum, 1E-9, message:='Profile[0] maximum incorrect');
// AssertEquals_LREAL(0.12819874947134405, positionExtrema.Tmin, 1E-9, message:='Profile[0] Tmin incorrect');
AssertEquals_LREAL(25.57994474955607699940, positionExtrema.Minimum, 1E-9, message:='Profile[0] minimum incorrect');

positionExtrema := ruckig._profiles[1].positionExtrema();
AssertEquals_LREAL(0.00000000000000000000, positionExtrema.Tmax, 1E-9, message:='Profile[1] Tmax incorrect');
AssertEquals_LREAL(31.55963588984187140341, positionExtrema.Maximum, 1E-9, message:='Profile[1] maximum incorrect');
// AssertEquals_LREAL(0.12819874947134405, positionExtrema.Tmin, 1E-9, message:='Profile[1] Tmin incorrect');
AssertEquals_LREAL(-15.83091418217285806236, positionExtrema.Minimum, 1E-9, message:='Profile[1] minimum incorrect');

positionExtrema := ruckig._profiles[2].positionExtrema();
AssertEquals_LREAL(0.00000000000000000000, positionExtrema.Tmax, 1E-9, message:='Profile[2] Tmax incorrect');
AssertEquals_LREAL(-13.09422790776093847853, positionExtrema.Maximum, 1E-9, message:='Profile[2] maximum incorrect');
// AssertEquals_LREAL(0.12819874947134405, positionExtrema.Tmin, 1E-9, message:='Profile[2] Tmin incorrect');
// AssertEquals_LREAL(-48.94577744042891254139, positionExtrema.Minimum, 1E-9, message:='Profile[2] minimum incorrect');
   

TEST_FINISHED();
END_METHOD

METHOD Test_Trajectory_6
VAR_INST
  ruckig : Struckig.Otg(0.001, 3) := (
  
    Synchronization := SynchronizationType.TimeSync,        
    MaxVelocity := [ 2000.00000000000000000000, 2000.00000000000000000000, 2000.00000000000000000000 ],
    MaxAcceleration := [ 20000.00000000000000000000, 20000.00000000000000000000, 20000.00000000000000000000 ],
    MaxJerk := [ 800000.00000000000000000000, 800000.00000000000000000000, 800000.00000000000000000000 ],
    CurrentPosition := [ 34.87125433480801461883, -76.41743919954686248275, -14.51229957505336187751 ],
    CurrentVelocity := [ -351.47533977255477566359, -987.15940067026019733021, 806.52305687867078631825 ],
    CurrentAcceleration := [ 1479.98184028979630966205, 8781.04772240824968321249, -8054.60406117963975702878 ],
    TargetPosition := [ 89.75739755287582966048, -1.42163448044479423515, -1.45152739794252738648 ],
    TargetVelocity := [ 0.00000000000000000000, 0.00000000000000000000, 0.00000000000000000000 ],
    TargetAcceleration := [ 0.00000000000000000000, 0.00000000000000000000, 0.00000000000000000000 ]
  );
  
  positionExtrema : Struckig.PositionExtremaDesc;
END_VAR
TEST('Trajectory_6');

ruckig();

// Check total duration of profiles
AssertEquals_LREAL(Expected := 0.21185526251360681238, Actual := ruckig.Duration, DELTA := 1E-8, Message := 'Duration incorrect');

// Check duration for each phase
positionExtrema := ruckig._profiles[0].positionExtrema();
AssertEquals_LREAL(0.21185526251360681238, positionExtrema.Tmax, 1E-9, message:='Profile[0] Tmax incorrect');
AssertEquals_LREAL(89.75739755287582966048, positionExtrema.Maximum, 1E-9, message:='Profile[0] maximum incorrect');
AssertEquals_LREAL(0.02315002269963775672, positionExtrema.Tmin, 1E-9, message:='Profile[0] Tmin incorrect');
AssertEquals_LREAL(28.78538978510774271058, positionExtrema.Minimum, 1E-9, message:='Profile[0] minimum incorrect');

positionExtrema := ruckig._profiles[1].positionExtrema();
AssertEquals_LREAL(0.21185526251360681238, positionExtrema.Tmax, 1E-9, message:='Profile[1] Tmax incorrect');
AssertEquals_LREAL(-1.42163448044479423515, positionExtrema.Maximum, 1E-9, message:='Profile[1] maximum incorrect');
AssertEquals_LREAL(0.01402369034698968710, positionExtrema.Tmin, 1E-9, message:='Profile[1] Tmin incorrect');
AssertEquals_LREAL(-89.02987231727530570424, positionExtrema.Minimum, 1E-9, message:='Profile[1] minimum incorrect');

positionExtrema := ruckig._profiles[2].positionExtrema();
AssertEquals_LREAL(0.04895379271357422346, positionExtrema.Tmax, 1E-9, message:='Profile[2] Tmax incorrect');
AssertEquals_LREAL(5.32847853519255032495, positionExtrema.Maximum, 1E-9, message:='Profile[2] maximum incorrect');
AssertEquals_LREAL(0.00000000000000000000, positionExtrema.Tmin, 1E-9, message:='Profile[2] Tmin incorrect');
AssertEquals_LREAL(-14.51229957505336187751, positionExtrema.Minimum, 1E-9, message:='Profile[2] minimum incorrect');
   

TEST_FINISHED();
END_METHOD

METHOD Test_Trajectory_62
VAR_INST
  ruckig : Struckig.Otg(0.001, 3) := (
  
    Synchronization := SynchronizationType.TimeSync,        
    MaxVelocity := [ 2000.00000000000000000000, 2000.00000000000000000000, 2000.00000000000000000000 ],
    MaxAcceleration := [ 20000.00000000000000000000, 20000.00000000000000000000, 20000.00000000000000000000 ],
    MaxJerk := [ 800000.00000000000000000000, 800000.00000000000000000000, 800000.00000000000000000000 ],
    CurrentPosition := [ 12.59051349490785298713, 2.34116410267218100216, -83.91521339841989401975 ],
    CurrentVelocity := [ -551.49352374949262411974, 694.95621845049936382566, -934.69209805013122149830 ],
    CurrentAcceleration := [ -5149.29503825546817097347, -9527.17655518820902216248, -9641.67382351083688263316 ],
    TargetPosition := [ -69.43235683496359911260, 5.95471336539937112775, -76.71462247839342296629 ],
    TargetVelocity := [ 0.00000000000000000000, 0.00000000000000000000, 0.00000000000000000000 ],
    TargetAcceleration := [ 0.00000000000000000000, 0.00000000000000000000, 0.00000000000000000000 ]
  );
  
  positionExtrema : Struckig.PositionExtremaDesc;
END_VAR
TEST('Trajectory_62');

ruckig();

// Check total duration of profiles
AssertEquals_LREAL(Expected := 0.19541920510428964497, Actual := ruckig.Duration, DELTA := 1E-8, Message := 'Duration incorrect');

// Check duration for each phase
positionExtrema := ruckig._profiles[0].positionExtrema();
AssertEquals_LREAL(0.00000000000000000000, positionExtrema.Tmax, 1E-9, message:='Profile[0] Tmax incorrect');
AssertEquals_LREAL(12.59051349490785298713, positionExtrema.Maximum, 1E-9, message:='Profile[0] maximum incorrect');
AssertEquals_LREAL(0.19541920510428961721, positionExtrema.Tmin, 1E-9, message:='Profile[0] Tmin incorrect');
AssertEquals_LREAL(-69.43235683496359911260, positionExtrema.Minimum, 1E-9, message:='Profile[0] minimum incorrect');

positionExtrema := ruckig._profiles[1].positionExtrema();
AssertEquals_LREAL(0.04065736745126265206, positionExtrema.Tmax, 1E-9, message:='Profile[1] Tmax incorrect');
AssertEquals_LREAL(16.73830873177616496150, positionExtrema.Maximum, 1E-9, message:='Profile[1] maximum incorrect');
AssertEquals_LREAL(0.00000000000000000000, positionExtrema.Tmin, 1E-9, message:='Profile[1] Tmin incorrect');
AssertEquals_LREAL(2.34116410267218100216, positionExtrema.Minimum, 1E-9, message:='Profile[1] minimum incorrect');

positionExtrema := ruckig._profiles[2].positionExtrema();
AssertEquals_LREAL(0.19541920510428964497, positionExtrema.Tmax, 1E-9, message:='Profile[2] Tmax incorrect');
AssertEquals_LREAL(-76.71462247839342296629, positionExtrema.Maximum, 1E-9, message:='Profile[2] maximum incorrect');
AssertEquals_LREAL(0.10355548042620135729, positionExtrema.Tmin, 1E-9, message:='Profile[2] Tmin incorrect');
AssertEquals_LREAL(-123.55479709285413036923, positionExtrema.Minimum, 1E-9, message:='Profile[2] minimum incorrect');
   

TEST_FINISHED();
END_METHOD

METHOD Test_Trajectory_64
VAR_INST
  ruckig : Struckig.Otg(0.001, 3) := (
  
    Synchronization := SynchronizationType.TimeSync,        
    MaxVelocity := [ 2000.00000000000000000000, 2000.00000000000000000000, 2000.00000000000000000000 ],
    MaxAcceleration := [ 20000.00000000000000000000, 20000.00000000000000000000, 20000.00000000000000000000 ],
    MaxJerk := [ 800000.00000000000000000000, 800000.00000000000000000000, 800000.00000000000000000000 ],
    CurrentPosition := [ 84.12964321952199497900, 15.09477787023756434337, 10.23674324179428651860 ],
    CurrentVelocity := [ -970.87417203950269595225, -928.12491864862022339366, 286.06399288670468195050 ],
    CurrentAcceleration := [ 4961.60497362833666556980, 5135.12661885897978208959, 79.48669035600505594630 ],
    TargetPosition := [ -30.09864175377319384097, 39.92408869665283077666, 24.17762560090359613696 ],
    TargetVelocity := [ 0.00000000000000000000, 0.00000000000000000000, 0.00000000000000000000 ],
    TargetAcceleration := [ 0.00000000000000000000, 0.00000000000000000000, 0.00000000000000000000 ]
  );
  
  positionExtrema : Struckig.PositionExtremaDesc;
END_VAR
TEST('Trajectory_64');

ruckig();

// Check total duration of profiles
AssertEquals_LREAL(Expected := 0.17167999763375443867, Actual := ruckig.Duration, DELTA := 1E-8, Message := 'Duration incorrect');

// Check duration for each phase
positionExtrema := ruckig._profiles[0].positionExtrema();
AssertEquals_LREAL(0.00000000000000000000, positionExtrema.Tmax, 1E-9, message:='Profile[0] Tmax incorrect');
AssertEquals_LREAL(84.12964321952199497900, positionExtrema.Maximum, 1E-9, message:='Profile[0] maximum incorrect');
AssertEquals_LREAL(0.17167999763375441091, positionExtrema.Tmin, 1E-9, message:='Profile[0] Tmin incorrect');
AssertEquals_LREAL(-30.09864175377319384097, positionExtrema.Minimum, 1E-9, message:='Profile[0] minimum incorrect');

positionExtrema := ruckig._profiles[1].positionExtrema();
AssertEquals_LREAL(0.17167999763375443867, positionExtrema.Tmax, 1E-9, message:='Profile[1] Tmax incorrect');
AssertEquals_LREAL(39.92408869665283077666, positionExtrema.Maximum, 1E-9, message:='Profile[1] maximum incorrect');
AssertEquals_LREAL(0.08124569148055139911, positionExtrema.Tmin, 1E-9, message:='Profile[1] Tmin incorrect');
AssertEquals_LREAL(-4.66763872582565753078, positionExtrema.Minimum, 1E-9, message:='Profile[1] minimum incorrect');

positionExtrema := ruckig._profiles[2].positionExtrema();
AssertEquals_LREAL(0.17167999763375443867, positionExtrema.Tmax, 1E-9, message:='Profile[2] Tmax incorrect');
AssertEquals_LREAL(24.17762560090359613696, positionExtrema.Maximum, 1E-9, message:='Profile[2] maximum incorrect');
AssertEquals_LREAL(0.00000000000000000000, positionExtrema.Tmin, 1E-9, message:='Profile[2] Tmin incorrect');
AssertEquals_LREAL(10.23674324179428651860, positionExtrema.Minimum, 1E-9, message:='Profile[2] minimum incorrect');
   

TEST_FINISHED();
END_METHOD

METHOD Test_Trajectory_65
VAR_INST
  ruckig : Struckig.Otg(0.001, 3) := (
  
    Synchronization := SynchronizationType.TimeSync,        
    MaxVelocity := [ 2000.00000000000000000000, 2000.00000000000000000000, 2000.00000000000000000000 ],
    MaxAcceleration := [ 20000.00000000000000000000, 20000.00000000000000000000, 20000.00000000000000000000 ],
    MaxJerk := [ 800000.00000000000000000000, 800000.00000000000000000000, 800000.00000000000000000000 ],
    CurrentPosition := [ 33.17628426446438538733, 50.00168428476928283999, 61.64263417164463021436 ],
    CurrentVelocity := [ -519.65995269471272877126, 66.93100559795539084007, -520.26416261644567384792 ],
    CurrentAcceleration := [ 3662.19439283437168342061, -8995.68879146701328863855, 4153.78894930269962060265 ],
    TargetPosition := [ 68.69261284366797326584, -66.97490772805458902894, -0.91414242050534255668 ],
    TargetVelocity := [ 0.00000000000000000000, 0.00000000000000000000, 0.00000000000000000000 ],
    TargetAcceleration := [ 0.00000000000000000000, 0.00000000000000000000, 0.00000000000000000000 ]
  );
  
  positionExtrema : Struckig.PositionExtremaDesc;
END_VAR
TEST('Trajectory_65');

ruckig();

// Check total duration of profiles
AssertEquals_LREAL(Expected := 0.17505526811503621665, Actual := ruckig.Duration, DELTA := 1E-8, Message := 'Duration incorrect');

// Check duration for each phase
positionExtrema := ruckig._profiles[0].positionExtrema();
AssertEquals_LREAL(0.17505526811503624440, positionExtrema.Tmax, 1E-9, message:='Profile[0] Tmax incorrect');
AssertEquals_LREAL(68.69261284366797326584, positionExtrema.Maximum, 1E-9, message:='Profile[0] maximum incorrect');
AssertEquals_LREAL(0.04377678309027987352, positionExtrema.Tmin, 1E-9, message:='Profile[0] Tmin incorrect');
AssertEquals_LREAL(23.42380651880664998998, positionExtrema.Minimum, 1E-9, message:='Profile[0] minimum incorrect');

positionExtrema := ruckig._profiles[1].positionExtrema();
AssertEquals_LREAL(0.00589507367218594907, positionExtrema.Tmax, 1E-9, message:='Profile[1] Tmax incorrect');
AssertEquals_LREAL(50.21262355411419520124, positionExtrema.Maximum, 1E-9, message:='Profile[1] maximum incorrect');
AssertEquals_LREAL(0.17505526811503621665, positionExtrema.Tmin, 1E-9, message:='Profile[1] Tmin incorrect');
AssertEquals_LREAL(-66.97490772805458902894, positionExtrema.Minimum, 1E-9, message:='Profile[1] minimum incorrect');

positionExtrema := ruckig._profiles[2].positionExtrema();
AssertEquals_LREAL(0.00000000000000000000, positionExtrema.Tmax, 1E-9, message:='Profile[2] Tmax incorrect');
AssertEquals_LREAL(61.64263417164463021436, positionExtrema.Maximum, 1E-9, message:='Profile[2] maximum incorrect');
AssertEquals_LREAL(0.17505526750468464181, positionExtrema.Tmin, 1E-9, message:='Profile[2] Tmin incorrect');
AssertEquals_LREAL(-0.91414242050535987616, positionExtrema.Minimum, 1E-9, message:='Profile[2] minimum incorrect');
   

TEST_FINISHED();
END_METHOD

METHOD Test_Trajectory_68
VAR_INST
  ruckig : Struckig.Otg(0.001, 3) := (
  
    Synchronization := SynchronizationType.TimeSync,        
    MaxVelocity := [ 2000.00000000000000000000, 2000.00000000000000000000, 2000.00000000000000000000 ],
    MaxAcceleration := [ 20000.00000000000000000000, 20000.00000000000000000000, 20000.00000000000000000000 ],
    MaxJerk := [ 800000.00000000000000000000, 800000.00000000000000000000, 800000.00000000000000000000 ],
    CurrentPosition := [ 40.62614323446814523777, 62.35469594204587906461, 24.25299098284108367807 ],
    CurrentVelocity := [ 953.39433299337724747602, 990.56715267728145590809, -738.17109364107295732538 ],
    CurrentAcceleration := [ 3444.24110064584601786919, 3257.77518810100627888460, 851.25313620111410273239 ],
    TargetPosition := [ -19.90968527499555307259, -93.17120052432892407523, -41.77005066216172934901 ],
    TargetVelocity := [ 0.00000000000000000000, 0.00000000000000000000, 0.00000000000000000000 ],
    TargetAcceleration := [ 0.00000000000000000000, 0.00000000000000000000, 0.00000000000000000000 ]
  );
  
  positionExtrema : Struckig.PositionExtremaDesc;
END_VAR
TEST('Trajectory_68');

ruckig();

// Check total duration of profiles
AssertEquals_LREAL(Expected := 0.27894619941724319023, Actual := ruckig.Duration, DELTA := 1E-8, Message := 'Duration incorrect');

// Check duration for each phase
positionExtrema := ruckig._profiles[0].positionExtrema();
AssertEquals_LREAL(0.08122133382222911091, positionExtrema.Tmax, 1E-9, message:='Profile[0] Tmax incorrect');
AssertEquals_LREAL(76.63857184314483106391, positionExtrema.Maximum, 1E-9, message:='Profile[0] maximum incorrect');
AssertEquals_LREAL(0.27894619941724324574, positionExtrema.Tmin, 1E-9, message:='Profile[0] Tmin incorrect');
AssertEquals_LREAL(-19.90968527499555307259, positionExtrema.Minimum, 1E-9, message:='Profile[0] minimum incorrect');

positionExtrema := ruckig._profiles[1].positionExtrema();
AssertEquals_LREAL(0.02907221898512625524, positionExtrema.Tmax, 1E-9, message:='Profile[1] Tmax incorrect');
AssertEquals_LREAL(89.25318532542951288633, positionExtrema.Maximum, 1E-9, message:='Profile[1] maximum incorrect');
AssertEquals_LREAL(0.27894619941724319023, positionExtrema.Tmin, 1E-9, message:='Profile[1] Tmin incorrect');
AssertEquals_LREAL(-93.17120052432892407523, positionExtrema.Minimum, 1E-9, message:='Profile[1] minimum incorrect');

positionExtrema := ruckig._profiles[2].positionExtrema();
AssertEquals_LREAL(0.00000000000000000000, positionExtrema.Tmax, 1E-9, message:='Profile[2] Tmax incorrect');
AssertEquals_LREAL(24.25299098284108367807, positionExtrema.Maximum, 1E-9, message:='Profile[2] maximum incorrect');
AssertEquals_LREAL(0.27894619941724324574, positionExtrema.Tmin, 1E-9, message:='Profile[2] Tmin incorrect');
AssertEquals_LREAL(-41.77005066216172934901, positionExtrema.Minimum, 1E-9, message:='Profile[2] minimum incorrect');
   

TEST_FINISHED();
END_METHOD

METHOD Test_Trajectory_7
VAR_INST
  ruckig : Struckig.Otg(0.001, 3) := (
  
    Synchronization := SynchronizationType.TimeSync,        
    MaxVelocity := [ 2000.00000000000000000000, 2000.00000000000000000000, 2000.00000000000000000000 ],
    MaxAcceleration := [ 20000.00000000000000000000, 20000.00000000000000000000, 20000.00000000000000000000 ],
    MaxJerk := [ 800000.00000000000000000000, 800000.00000000000000000000, 800000.00000000000000000000 ],
    CurrentPosition := [ -12.40730451188392180484, -80.83422386552678062799, 12.57670349433081469215 ],
    CurrentVelocity := [ 265.90445653002484505123, 357.90733431729245239694, 18.46515886490806224174 ],
    CurrentAcceleration := [ -2167.27013269919098092942, 949.55886260518127528485, 2528.49090058209003473166 ],
    TargetPosition := [ -97.77133953691699730371, -53.09340578221126349945, -63.96892666434119689711 ],
    TargetVelocity := [ 0.00000000000000000000, 0.00000000000000000000, 0.00000000000000000000 ],
    TargetAcceleration := [ 0.00000000000000000000, 0.00000000000000000000, 0.00000000000000000000 ]
  );
  
  positionExtrema : Struckig.PositionExtremaDesc;
END_VAR
TEST('Trajectory_7');

ruckig();

// Check total duration of profiles
AssertEquals_LREAL(Expected := 0.17206395017599335207, Actual := ruckig.Duration, DELTA := 1E-8, Message := 'Duration incorrect');

// Check duration for each phase
positionExtrema := ruckig._profiles[0].positionExtrema();
AssertEquals_LREAL(0.02229091233412601111, positionExtrema.Tmax, 1E-9, message:='Profile[0] Tmax incorrect');
AssertEquals_LREAL(-8.49529533349170762335, positionExtrema.Maximum, 1E-9, message:='Profile[0] maximum incorrect');
AssertEquals_LREAL(0.17206395017599335207, positionExtrema.Tmin, 1E-9, message:='Profile[0] Tmin incorrect');
AssertEquals_LREAL(-97.77133953691699730371, positionExtrema.Minimum, 1E-9, message:='Profile[0] minimum incorrect');

positionExtrema := ruckig._profiles[1].positionExtrema();
AssertEquals_LREAL(0.17206395017599335207, positionExtrema.Tmax, 1E-9, message:='Profile[1] Tmax incorrect');
AssertEquals_LREAL(-53.09340578221126349945, positionExtrema.Maximum, 1E-9, message:='Profile[1] maximum incorrect');
AssertEquals_LREAL(0.00000000000000000000, positionExtrema.Tmin, 1E-9, message:='Profile[1] Tmin incorrect');
AssertEquals_LREAL(-80.83422386552678062799, positionExtrema.Minimum, 1E-9, message:='Profile[1] minimum incorrect');

positionExtrema := ruckig._profiles[2].positionExtrema();
AssertEquals_LREAL(0.01065410250964578427, positionExtrema.Tmax, 1E-9, message:='Profile[2] Tmax incorrect');
AssertEquals_LREAL(12.75569141626643698828, positionExtrema.Maximum, 1E-9, message:='Profile[2] maximum incorrect');
AssertEquals_LREAL(0.17206395017599335207, positionExtrema.Tmin, 1E-9, message:='Profile[2] Tmin incorrect');
AssertEquals_LREAL(-63.96892666434119689711, positionExtrema.Minimum, 1E-9, message:='Profile[2] minimum incorrect');
   

TEST_FINISHED();
END_METHOD

END_FUNCTION_BLOCK

// ---- POUs/TargetPosAccTest.TcPOU
FUNCTION_BLOCK TargetPosAccTest EXTENDS TcUnit.FB_TestSuite
VAR
  ruckig : Struckig.Otg(0.001, 3) := (
  
    Synchronization := SynchronizationType.TimeSync,        
    MaxVelocity := [ 2000.00000000000000000000, 2000.00000000000000000000, 2000.00000000000000000000 ],
    MaxAcceleration := [ 20000.00000000000000000000, 20000.00000000000000000000, 20000.00000000000000000000 ],
    MaxJerk := [ 800000.00000000000000000000, 800000.00000000000000000000, 800000.00000000000000000000 ],
    CurrentPosition := [ 48.86656216713086564596, 31.55963588984187140341, -13.09422790776093847853 ],
    CurrentVelocity := [ -274.21841080128081102885, -440.94461360926254656079, -764.75678162210920163488 ],
    CurrentAcceleration := [ -1478.09700836416959646158, 686.79611869591644790489, -9263.72976579731221136171 ],
    TargetPosition := [ 25.57994474955607699940, -15.83091418217283319336, -38.97164514571973370494 ],
    TargetVelocity := [ 0.00000000000000000000, 0.00000000000000000000, 0.00000000000000000000 ],
    TargetAcceleration := [ 0.00000000000000000000, 0.00000000000000000000, 0.00000000000000000000 ]
  );
  
  positionExtrema : Struckig.PositionExtremaDesc;  
END_VAR

Test_Trajectory_HasTargetAcceleration_8();
Test_Trajectory_HasTargetAcceleration_18();
Test_Trajectory_HasTargetAcceleration_26();
Test_Trajectory_HasTargetAcceleration_29();
Test_Trajectory_HasTargetAcceleration_39();
Test_Trajectory_HasTargetAcceleration_43();
Test_Trajectory_HasTargetAcceleration_50();
Test_Trajectory_HasTargetAcceleration_57();
Test_Trajectory_HasTargetAcceleration_58();
Test_Trajectory_HasTargetAcceleration_63();
Test_Trajectory_HasTargetAcceleration_67();

METHOD Test_Trajectory_HasTargetAcceleration_18
VAR_INST
  ruckig : Struckig.Otg(0.001, 3) := (
  
    Synchronization := SynchronizationType.TimeSync,        
    MaxVelocity := [ 2000.00000000000000000000, 2000.00000000000000000000, 2000.00000000000000000000 ],
    MaxAcceleration := [ 20000.00000000000000000000, 20000.00000000000000000000, 20000.00000000000000000000 ],
    MaxJerk := [ 800000.00000000000000000000, 800000.00000000000000000000, 800000.00000000000000000000 ],
    CurrentPosition := [ 22.29044197833951557186, -39.95859595632313698843, 54.11499073315658847605 ],
    CurrentVelocity := [ 553.01033394001592569111, 267.36329442224518970761, 895.38647163815880958282 ],
    CurrentAcceleration := [ 4077.95591124392740312032, -4124.70260840723312867340, -6307.27396104388935782481 ],
    TargetPosition := [ 19.06397199072051762414, 8.08665977239270716836, -61.80722661584501054222 ],
    TargetVelocity := [ 0.00000000000000000000, 0.00000000000000000000, 0.00000000000000000000 ],
    TargetAcceleration := [ -663.32888732782430452062, 140.67534288890783500392, 211.50762532936892057478 ]
  );
  
  positionExtrema : Struckig.PositionExtremaDesc;
END_VAR
TEST('Trajectory_HasTargetAcceleration_18');

ruckig();

// Check total duration of profiles
AssertEquals_LREAL(Expected := 0.23288436093144340711, Actual := ruckig.Duration, DELTA := 1E-8, Message := 'Duration incorrect');

// Check duration for each phase
positionExtrema := ruckig._profiles[0].positionExtrema();
AssertEquals_LREAL(0.04687484204301414770, positionExtrema.Tmax, 1E-9, message:='Profile[0] Tmax incorrect');
AssertEquals_LREAL(39.64467835267222994844, positionExtrema.Maximum, 1E-9, message:='Profile[0] maximum incorrect');
AssertEquals_LREAL(0.23122603871312383261, positionExtrema.Tmin, 1E-9, message:='Profile[0] Tmin incorrect');
AssertEquals_LREAL(19.06366796137865549099, positionExtrema.Minimum, 1E-9, message:='Profile[0] minimum incorrect');

positionExtrema := ruckig._profiles[1].positionExtrema();
AssertEquals_LREAL(0.23253267257422116643, positionExtrema.Tmax, 1E-9, message:='Profile[1] Tmax incorrect');
AssertEquals_LREAL(8.08666267229066093591, positionExtrema.Maximum, 1E-9, message:='Profile[1] maximum incorrect');
AssertEquals_LREAL(0.00000000000000000000, positionExtrema.Tmin, 1E-9, message:='Profile[1] Tmin incorrect');
AssertEquals_LREAL(-39.95859595632313698843, positionExtrema.Minimum, 1E-9, message:='Profile[1] minimum incorrect');

positionExtrema := ruckig._profiles[2].positionExtrema();
AssertEquals_LREAL(0.01711590754869513759, positionExtrema.Tmax, 1E-9, message:='Profile[2] Tmax incorrect');
AssertEquals_LREAL(67.84791417376290212360, positionExtrema.Maximum, 1E-9, message:='Profile[2] maximum incorrect');
AssertEquals_LREAL(0.23288436093144340711, positionExtrema.Tmin, 1E-9, message:='Profile[2] Tmin incorrect');
AssertEquals_LREAL(-61.80722661584501054222, positionExtrema.Minimum, 1E-9, message:='Profile[2] minimum incorrect');
   

TEST_FINISHED();
END_METHOD

METHOD Test_Trajectory_HasTargetAcceleration_26
VAR_INST
  ruckig : Struckig.Otg(0.001, 3) := (
  
    Synchronization := SynchronizationType.TimeSync,        
    MaxVelocity := [ 2000.00000000000000000000, 2000.00000000000000000000, 2000.00000000000000000000 ],
    MaxAcceleration := [ 20000.00000000000000000000, 20000.00000000000000000000, 20000.00000000000000000000 ],
    MaxJerk := [ 800000.00000000000000000000, 800000.00000000000000000000, 800000.00000000000000000000 ],
    CurrentPosition := [ 77.39232107651710634855, -63.03832121402539456767, 50.64263565514380616150 ],
    CurrentVelocity := [ 390.27238163421588978963, -873.49794562195870639698, 981.87086783538688905537 ],
    CurrentAcceleration := [ 7745.26876878265466075391, -2376.69313379117920703720, 3911.92493779323558555916 ],
    TargetPosition := [ -47.12017227692884091539, 44.57407397341043520100, 81.30379250690350545483 ],
    TargetVelocity := [ 0.00000000000000000000, 0.00000000000000000000, 0.00000000000000000000 ],
    TargetAcceleration := [ 543.91131759469612916291, 821.67345447350203357928, 930.33404428054154777783 ]
  );
  
  positionExtrema : Struckig.PositionExtremaDesc;
END_VAR
TEST('Trajectory_HasTargetAcceleration_26');

ruckig();

// Check total duration of profiles
AssertEquals_LREAL(Expected := 0.24230324879908460289, Actual := ruckig.Duration, DELTA := 1E-8, Message := 'Duration incorrect');

// Check duration for each phase
positionExtrema := ruckig._profiles[0].positionExtrema();
AssertEquals_LREAL(0.03468158596097831864, positionExtrema.Tmax, 1E-9, message:='Profile[0] Tmax incorrect');
AssertEquals_LREAL(90.02357999691733425607, positionExtrema.Maximum, 1E-9, message:='Profile[0] maximum incorrect');
AssertEquals_LREAL(0.24230324879908460289, positionExtrema.Tmin, 1E-9, message:='Profile[0] Tmin incorrect');
AssertEquals_LREAL(-47.12017227692884091539, positionExtrema.Minimum, 1E-9, message:='Profile[0] minimum incorrect');

positionExtrema := ruckig._profiles[1].positionExtrema();
AssertEquals_LREAL(0.24024906516290109315, positionExtrema.Tmax, 1E-9, message:='Profile[1] Tmax incorrect');
AssertEquals_LREAL(44.57465183860438884267, positionExtrema.Maximum, 1E-9, message:='Profile[1] maximum incorrect');
AssertEquals_LREAL(0.02797086641723897649, positionExtrema.Tmin, 1E-9, message:='Profile[1] Tmin incorrect');
AssertEquals_LREAL(-85.48273497475497606501, positionExtrema.Minimum, 1E-9, message:='Profile[1] minimum incorrect');

positionExtrema := ruckig._profiles[2].positionExtrema();
AssertEquals_LREAL(0.06985653728563799569, positionExtrema.Tmax, 1E-9, message:='Profile[2] Tmax incorrect');
AssertEquals_LREAL(92.06916456436438522815, positionExtrema.Maximum, 1E-9, message:='Profile[2] maximum incorrect');
AssertEquals_LREAL(0.00000000000000000000, positionExtrema.Tmin, 1E-9, message:='Profile[2] Tmin incorrect');
AssertEquals_LREAL(50.64263565514380616150, positionExtrema.Minimum, 1E-9, message:='Profile[2] minimum incorrect');
   

TEST_FINISHED();
END_METHOD

METHOD Test_Trajectory_HasTargetAcceleration_29
VAR_INST
  ruckig : Struckig.Otg(0.001, 3) := (
  
    Synchronization := SynchronizationType.TimeSync,        
    MaxVelocity := [ 2000.00000000000000000000, 2000.00000000000000000000, 2000.00000000000000000000 ],
    MaxAcceleration := [ 20000.00000000000000000000, 20000.00000000000000000000, 20000.00000000000000000000 ],
    MaxJerk := [ 800000.00000000000000000000, 800000.00000000000000000000, 800000.00000000000000000000 ],
    CurrentPosition := [ 44.91183232377716194605, 20.60848326549906062155, -39.18243853552834110587 ],
    CurrentVelocity := [ 56.12947053833636346099, 974.84045859192679017724, 288.91800445440071598568 ],
    CurrentAcceleration := [ -7725.89726821354634012096, 1120.94279215741516964044, 3716.25460982452932512388 ],
    TargetPosition := [ 82.62783593756236655281, -34.57308232880984633084, 42.27769995179082229697 ],
    TargetVelocity := [ 0.00000000000000000000, 0.00000000000000000000, 0.00000000000000000000 ],
    TargetAcceleration := [ -115.18831231873787146469, 604.54144453707817774557, -488.03361084610719444754 ]
  );
  
  positionExtrema : Struckig.PositionExtremaDesc;
END_VAR
TEST('Trajectory_HasTargetAcceleration_29');

ruckig();

// Check total duration of profiles
AssertEquals_LREAL(Expected := 0.21276205615654666947, Actual := ruckig.Duration, DELTA := 1E-8, Message := 'Duration incorrect');

// Check duration for each phase
positionExtrema := ruckig._profiles[0].positionExtrema();
AssertEquals_LREAL(0.21276205615654666947, positionExtrema.Tmax, 1E-9, message:='Profile[0] Tmax incorrect');
AssertEquals_LREAL(82.62783593756236655281, positionExtrema.Maximum, 1E-9, message:='Profile[0] maximum incorrect');
AssertEquals_LREAL(0.00000000000000000000, positionExtrema.Tmin, 1E-9, message:='Profile[0] Tmin incorrect');
AssertEquals_LREAL(44.91183232377716194605, positionExtrema.Minimum, 1E-9, message:='Profile[0] minimum incorrect');

positionExtrema := ruckig._profiles[1].positionExtrema();
AssertEquals_LREAL(0.02640117849019677290, positionExtrema.Tmax, 1E-9, message:='Profile[1] Tmax incorrect');
AssertEquals_LREAL(44.28245347329226433430, positionExtrema.Maximum, 1E-9, message:='Profile[1] maximum incorrect');
AssertEquals_LREAL(0.21276205615654666947, positionExtrema.Tmin, 1E-9, message:='Profile[1] Tmin incorrect');
AssertEquals_LREAL(-34.57308232880984633084, positionExtrema.Minimum, 1E-9, message:='Profile[1] minimum incorrect');

positionExtrema := ruckig._profiles[2].positionExtrema();
AssertEquals_LREAL(0.21276205615654666947, positionExtrema.Tmax, 1E-9, message:='Profile[2] Tmax incorrect');
AssertEquals_LREAL(42.27769995179082229697, positionExtrema.Maximum, 1E-9, message:='Profile[2] maximum incorrect');
AssertEquals_LREAL(0.00000000000000000000, positionExtrema.Tmin, 1E-9, message:='Profile[2] Tmin incorrect');
AssertEquals_LREAL(-39.18243853552834110587, positionExtrema.Minimum, 1E-9, message:='Profile[2] minimum incorrect');
   

TEST_FINISHED();
END_METHOD

METHOD Test_Trajectory_HasTargetAcceleration_37
VAR_INST
  ruckig : Struckig.Otg(0.001, 3) := (
  
    Synchronization := SynchronizationType.TimeSync,        
    MaxVelocity := [ 2000.00000000000000000000, 2000.00000000000000000000, 2000.00000000000000000000 ],
    MaxAcceleration := [ 20000.00000000000000000000, 20000.00000000000000000000, 20000.00000000000000000000 ],
    MaxJerk := [ 800000.00000000000000000000, 800000.00000000000000000000, 800000.00000000000000000000 ],
    CurrentPosition := [ 75.70258410717627839404, -31.81448222562724481577, -58.08554852109006816363 ],
    CurrentVelocity := [ 171.95882136884461033333, -584.70058950900761374214, 745.12321825604590230796 ],
    CurrentAcceleration := [ 5092.19654988173533638474, 7179.19572851603152230382, 1704.28450887377948674839 ],
    TargetPosition := [ 97.60417669221266123714, 88.97844242319803242935, -19.79432812800784802221 ],
    TargetVelocity := [ 0.00000000000000000000, 0.00000000000000000000, 0.00000000000000000000 ],
    TargetAcceleration := [ 983.95730849860865419032, -389.38723727042054179037, -311.43162034307158592128 ]
  );
  
  positionExtrema : Struckig.PositionExtremaDesc;
END_VAR
TEST('Trajectory_HasTargetAcceleration_37');

ruckig();

// Check total duration of profiles
AssertEquals_LREAL(Expected := 0.21113509394885510151, Actual := ruckig.Duration, DELTA := 1E-8, Message := 'Duration incorrect');

// Check duration for each phase
positionExtrema := ruckig._profiles[0].positionExtrema();
AssertEquals_LREAL(0.20867520067760855773, positionExtrema.Tmax, 1E-9, message:='Profile[0] Tmax incorrect');
AssertEquals_LREAL(97.60516902544232209493, positionExtrema.Maximum, 1E-9, message:='Profile[0] maximum incorrect');
AssertEquals_LREAL(0.00000000000000000000, positionExtrema.Tmin, 1E-9, message:='Profile[0] Tmin incorrect');
AssertEquals_LREAL(75.70258410717627839404, positionExtrema.Minimum, 1E-9, message:='Profile[0] minimum incorrect');

positionExtrema := ruckig._profiles[1].positionExtrema();
AssertEquals_LREAL(0.21113509394885510151, positionExtrema.Tmax, 1E-9, message:='Profile[1] Tmax incorrect');
AssertEquals_LREAL(88.97844242319803242935, positionExtrema.Maximum, 1E-9, message:='Profile[1] maximum incorrect');
AssertEquals_LREAL(0.01602600533935496022, positionExtrema.Tmin, 1E-9, message:='Profile[1] Tmin incorrect');
AssertEquals_LREAL(-39.71416974486287898571, positionExtrema.Minimum, 1E-9, message:='Profile[1] minimum incorrect');

positionExtrema := ruckig._profiles[2].positionExtrema();
AssertEquals_LREAL(0.21113509394885504600, positionExtrema.Tmax, 1E-9, message:='Profile[2] Tmax incorrect');
AssertEquals_LREAL(-19.79432812800784091678, positionExtrema.Maximum, 1E-9, message:='Profile[2] maximum incorrect');
AssertEquals_LREAL(0.00000000000000000000, positionExtrema.Tmin, 1E-9, message:='Profile[2] Tmin incorrect');
AssertEquals_LREAL(-58.08554852109006816363, positionExtrema.Minimum, 1E-9, message:='Profile[2] minimum incorrect');
   

TEST_FINISHED();
END_METHOD

METHOD Test_Trajectory_HasTargetAcceleration_39
VAR_INST
  ruckig : Struckig.Otg(0.001, 3) := (
  
    Synchronization := SynchronizationType.TimeSync,        
    MaxVelocity := [ 2000.00000000000000000000, 2000.00000000000000000000, 2000.00000000000000000000 ],
    MaxAcceleration := [ 20000.00000000000000000000, 20000.00000000000000000000, 20000.00000000000000000000 ],
    MaxJerk := [ 800000.00000000000000000000, 800000.00000000000000000000, 800000.00000000000000000000 ],
    CurrentPosition := [ -21.93974605417949419461, -18.49856402298217972202, -96.65992156980888694306 ],
    CurrentVelocity := [ 560.92968123589912465832, -454.79210991651348194864, -556.36905002756998328550 ],
    CurrentAcceleration := [ 6747.73447463338743546046, 9628.82123479624351602979, 5462.73061834566397010349 ],
    TargetPosition := [ -36.27372063241573840742, 69.45477693939508867516, -56.03831440156044152445 ],
    TargetVelocity := [ 0.00000000000000000000, 0.00000000000000000000, 0.00000000000000000000 ],
    TargetAcceleration := [ 228.31394350642813151353, -518.68886336123591718206, -694.01647177787629061640 ]
  );
  
  positionExtrema : Struckig.PositionExtremaDesc;
END_VAR
TEST('Trajectory_HasTargetAcceleration_39');

ruckig();

// Check total duration of profiles
AssertEquals_LREAL(Expected := 0.17804896497402217248, Actual := ruckig.Duration, DELTA := 1E-8, Message := 'Duration incorrect');

// Check duration for each phase
positionExtrema := ruckig._profiles[0].positionExtrema();
AssertEquals_LREAL(0.05596801189631349371, positionExtrema.Tmax, 1E-9, message:='Profile[0] Tmax incorrect');
AssertEquals_LREAL(-1.82711489240683677693, positionExtrema.Maximum, 1E-9, message:='Profile[0] maximum incorrect');
AssertEquals_LREAL(0.17804896497402203370, positionExtrema.Tmin, 1E-9, message:='Profile[0] Tmin incorrect');
AssertEquals_LREAL(-36.27372063241574551284, positionExtrema.Minimum, 1E-9, message:='Profile[0] minimum incorrect');

positionExtrema := ruckig._profiles[1].positionExtrema();
AssertEquals_LREAL(0.17804896497402217248, positionExtrema.Tmax, 1E-9, message:='Profile[1] Tmax incorrect');
AssertEquals_LREAL(69.45477693939508867516, positionExtrema.Maximum, 1E-9, message:='Profile[1] maximum incorrect');
AssertEquals_LREAL(0.01296397345650469532, positionExtrema.Tmin, 1E-9, message:='Profile[1] Tmin incorrect');
AssertEquals_LREAL(-23.29484015015810172144, positionExtrema.Minimum, 1E-9, message:='Profile[1] minimum incorrect');

positionExtrema := ruckig._profiles[2].positionExtrema();
AssertEquals_LREAL(0.17804896497402220024, positionExtrema.Tmax, 1E-9, message:='Profile[2] Tmax incorrect');
AssertEquals_LREAL(-56.03831440156044152445, positionExtrema.Maximum, 1E-9, message:='Profile[2] maximum incorrect');
AssertEquals_LREAL(0.04613976266622405592, positionExtrema.Tmin, 1E-9, message:='Profile[2] Tmin incorrect');
AssertEquals_LREAL(-106.33609120894020350079, positionExtrema.Minimum, 1E-9, message:='Profile[2] minimum incorrect');
   

TEST_FINISHED();
END_METHOD

METHOD Test_Trajectory_HasTargetAcceleration_42
VAR_INST
  ruckig : Struckig.Otg(0.001, 3) := (
  
    Synchronization := SynchronizationType.TimeSync,        
    MaxVelocity := [ 2000.00000000000000000000, 2000.00000000000000000000, 2000.00000000000000000000 ],
    MaxAcceleration := [ 20000.00000000000000000000, 20000.00000000000000000000, 20000.00000000000000000000 ],
    MaxJerk := [ 800000.00000000000000000000, 800000.00000000000000000000, 800000.00000000000000000000 ],
    CurrentPosition := [ 1.58314797372935345265, 90.58707779544036498010, 7.41484167737418431443 ],
    CurrentVelocity := [ 264.66369378964441239077, -967.86838256043972705811, 875.55912471800957064261 ],
    CurrentAcceleration := [ -5955.60883189429478079546, -8419.85921682317348313518, 8392.40723541911211214028 ],
    TargetPosition := [ -58.56616862494692554719, 73.15314018228875170280, 71.09694589628986705065 ],
    TargetVelocity := [ 0.00000000000000000000, 0.00000000000000000000, 0.00000000000000000000 ],
    TargetAcceleration := [ -714.77249466642297193175, -738.86959085233320365660, -949.40990195438507726067 ]
  );
  
  positionExtrema : Struckig.PositionExtremaDesc;
END_VAR
TEST('Trajectory_HasTargetAcceleration_42');

ruckig();

// Check total duration of profiles
AssertEquals_LREAL(Expected := 0.16824213942746521488, Actual := ruckig.Duration, DELTA := 1E-8, Message := 'Duration incorrect');

// Check duration for each phase
positionExtrema := ruckig._profiles[0].positionExtrema();
AssertEquals_LREAL(0.01755548896013213109, positionExtrema.Tmax, 1E-9, message:='Profile[0] Tmax incorrect');
AssertEquals_LREAL(4.59030121571332649921, positionExtrema.Maximum, 1E-9, message:='Profile[0] maximum incorrect');
AssertEquals_LREAL(0.16645520819079967501, positionExtrema.Tmin, 1E-9, message:='Profile[0] Tmin incorrect');
AssertEquals_LREAL(-58.56654901772477472832, positionExtrema.Minimum, 1E-9, message:='Profile[0] minimum incorrect');

positionExtrema := ruckig._profiles[1].positionExtrema();
AssertEquals_LREAL(0.00000000000000000000, positionExtrema.Tmax, 1E-9, message:='Profile[1] Tmax incorrect');
AssertEquals_LREAL(90.58707779544036498010, positionExtrema.Maximum, 1E-9, message:='Profile[1] maximum incorrect');
AssertEquals_LREAL(0.09014117386002259980, positionExtrema.Tmin, 1E-9, message:='Profile[1] Tmin incorrect');
AssertEquals_LREAL(45.07056608531748764790, positionExtrema.Minimum, 1E-9, message:='Profile[1] minimum incorrect');

positionExtrema := ruckig._profiles[2].positionExtrema();
AssertEquals_LREAL(0.13468422806677898818, positionExtrema.Tmax, 1E-9, message:='Profile[2] Tmax incorrect');
AssertEquals_LREAL(73.02284673044322005353, positionExtrema.Maximum, 1E-9, message:='Profile[2] maximum incorrect');
AssertEquals_LREAL(0.00000000000000000000, positionExtrema.Tmin, 1E-9, message:='Profile[2] Tmin incorrect');
AssertEquals_LREAL(7.41484167737418431443, positionExtrema.Minimum, 1E-9, message:='Profile[2] minimum incorrect');
   

TEST_FINISHED();
END_METHOD

METHOD Test_Trajectory_HasTargetAcceleration_43
VAR_INST
  ruckig : Struckig.Otg(0.001, 3) := (
  
    Synchronization := SynchronizationType.TimeSync,        
    MaxVelocity := [ 2000.00000000000000000000, 2000.00000000000000000000, 2000.00000000000000000000 ],
    MaxAcceleration := [ 20000.00000000000000000000, 20000.00000000000000000000, 20000.00000000000000000000 ],
    MaxJerk := [ 800000.00000000000000000000, 800000.00000000000000000000, 800000.00000000000000000000 ],
    CurrentPosition := [ 53.13739682938987130001, -22.44298053732963182938, -41.20042774153274223181 ],
    CurrentVelocity := [ -304.98663512538098530058, 35.02037430652057992120, 738.80078152761325327447 ],
    CurrentAcceleration := [ -7270.26712820171451312490, -845.41004591047749272548, -4566.56327336276262940373 ],
    TargetPosition := [ 81.86956314333414752582, 96.25424125499196748024, -65.78248687323761600965 ],
    TargetVelocity := [ 0.00000000000000000000, 0.00000000000000000000, 0.00000000000000000000 ],
    TargetAcceleration := [ -511.94239891635919548207, 447.91143210314089628810, -814.86235086373915237345 ]
  );
  
  positionExtrema : Struckig.PositionExtremaDesc;
END_VAR
TEST('Trajectory_HasTargetAcceleration_43');

ruckig();

// Check total duration of profiles
AssertEquals_LREAL(Expected := 0.18070492746146707419, Actual := ruckig.Duration, DELTA := 1E-8, Message := 'Duration incorrect');

// Check duration for each phase
positionExtrema := ruckig._profiles[0].positionExtrema();
AssertEquals_LREAL(0.18070492746146707419, positionExtrema.Tmax, 1E-9, message:='Profile[0] Tmax incorrect');
AssertEquals_LREAL(81.86956314333414752582, positionExtrema.Maximum, 1E-9, message:='Profile[0] maximum incorrect');
AssertEquals_LREAL(0.03408783391025214243, positionExtrema.Tmin, 1E-9, message:='Profile[0] Tmin incorrect');
AssertEquals_LREAL(43.79836178330638318812, positionExtrema.Minimum, 1E-9, message:='Profile[0] minimum incorrect');

positionExtrema := ruckig._profiles[1].positionExtrema();
AssertEquals_LREAL(0.17958514888120891140, positionExtrema.Tmax, 1E-9, message:='Profile[1] Tmax incorrect');
AssertEquals_LREAL(96.25433486131980487244, positionExtrema.Maximum, 1E-9, message:='Profile[1] maximum incorrect');
AssertEquals_LREAL(0.00000000000000000000, positionExtrema.Tmin, 1E-9, message:='Profile[1] Tmin incorrect');
AssertEquals_LREAL(-22.44298053732963182938, positionExtrema.Minimum, 1E-9, message:='Profile[1] minimum incorrect');

positionExtrema := ruckig._profiles[2].positionExtrema();
AssertEquals_LREAL(0.05355512909515708353, positionExtrema.Tmax, 1E-9, message:='Profile[2] Tmax incorrect');
AssertEquals_LREAL(-23.29997654589049815854, positionExtrema.Maximum, 1E-9, message:='Profile[2] maximum incorrect');
AssertEquals_LREAL(0.17866777158430743877, positionExtrema.Tmin, 1E-9, message:='Profile[2] Tmin incorrect');
AssertEquals_LREAL(-65.78305048691605350086, positionExtrema.Minimum, 1E-9, message:='Profile[2] minimum incorrect');
   

TEST_FINISHED();
END_METHOD

METHOD Test_Trajectory_HasTargetAcceleration_50
VAR_INST
  ruckig : Struckig.Otg(0.001, 3) := (
  
    Synchronization := SynchronizationType.TimeSync,        
    MaxVelocity := [ 2000.00000000000000000000, 2000.00000000000000000000, 2000.00000000000000000000 ],
    MaxAcceleration := [ 20000.00000000000000000000, 20000.00000000000000000000, 20000.00000000000000000000 ],
    MaxJerk := [ 800000.00000000000000000000, 800000.00000000000000000000, 800000.00000000000000000000 ],
    CurrentPosition := [ 46.92101107231894729921, -0.50374158461752926996, 29.71857774981103261780 ],
    CurrentVelocity := [ -825.06102637463254723116, 756.18378067008961807005, -198.33013045881875768828 ],
    CurrentAcceleration := [ -4766.41159160333245381480, -5907.94068977043207269162, -2476.07236462418222799897 ],
    TargetPosition := [ 23.42250735434379294020, 12.51307920714354793290, 2.55459165158602274914 ],
    TargetVelocity := [ 0.00000000000000000000, 0.00000000000000000000, 0.00000000000000000000 ],
    TargetAcceleration := [ -489.78938572767407322317, 603.07786572774739397573, -878.19166450623129094311 ]
  );
  
  positionExtrema : Struckig.PositionExtremaDesc;
END_VAR
TEST('Trajectory_HasTargetAcceleration_50');

ruckig();

// Check total duration of profiles
AssertEquals_LREAL(Expected := 0.12125503368046111619, Actual := ruckig.Duration, DELTA := 1E-8, Message := 'Duration incorrect');

// Check duration for each phase
positionExtrema := ruckig._profiles[0].positionExtrema();
AssertEquals_LREAL(0.00000000000000000000, positionExtrema.Tmax, 1E-9, message:='Profile[0] Tmax incorrect');
AssertEquals_LREAL(46.92101107231894729921, positionExtrema.Maximum, 1E-9, message:='Profile[0] maximum incorrect');
AssertEquals_LREAL(0.06087090854331475565, positionExtrema.Tmin, 1E-9, message:='Profile[0] Tmin incorrect');
AssertEquals_LREAL(14.37204891391303718251, positionExtrema.Minimum, 1E-9, message:='Profile[0] minimum incorrect');

positionExtrema := ruckig._profiles[1].positionExtrema();
AssertEquals_LREAL(0.04585205920535920243, positionExtrema.Tmax, 1E-9, message:='Profile[1] Tmax incorrect');
AssertEquals_LREAL(18.22432050158307603738, positionExtrema.Maximum, 1E-9, message:='Profile[1] maximum incorrect');
AssertEquals_LREAL(0.00000000000000000000, positionExtrema.Tmin, 1E-9, message:='Profile[1] Tmin incorrect');
AssertEquals_LREAL(-0.50374158461752926996, positionExtrema.Minimum, 1E-9, message:='Profile[1] minimum incorrect');

positionExtrema := ruckig._profiles[2].positionExtrema();
AssertEquals_LREAL(0.00000000000000000000, positionExtrema.Tmax, 1E-9, message:='Profile[2] Tmax incorrect');
AssertEquals_LREAL(29.71857774981103261780, positionExtrema.Maximum, 1E-9, message:='Profile[2] maximum incorrect');
AssertEquals_LREAL(0.11905955451919558730, positionExtrema.Tmin, 1E-9, message:='Profile[2] Tmin incorrect');
AssertEquals_LREAL(2.55388615210469760441, positionExtrema.Minimum, 1E-9, message:='Profile[2] minimum incorrect');
   

TEST_FINISHED();
END_METHOD

METHOD Test_Trajectory_HasTargetAcceleration_57
VAR_INST
  ruckig : Struckig.Otg(0.001, 3) := (
  
    Synchronization := SynchronizationType.TimeSync,        
    MaxVelocity := [ 2000.00000000000000000000, 2000.00000000000000000000, 2000.00000000000000000000 ],
    MaxAcceleration := [ 20000.00000000000000000000, 20000.00000000000000000000, 20000.00000000000000000000 ],
    MaxJerk := [ 800000.00000000000000000000, 800000.00000000000000000000, 800000.00000000000000000000 ],
    CurrentPosition := [ -41.78580401739355920654, -54.54341916085618890975, 0.34259842487062996952 ],
    CurrentVelocity := [ 281.70354130105670265038, 551.00897497765049592999, 302.83881748014778167999 ],
    CurrentAcceleration := [ 5924.00492373221095476765, 2065.11081253397605905775, 2773.66158712433571054135 ],
    TargetPosition := [ -35.55043245579965116576, 76.85926955676279703766, -20.12684108733012067205 ],
    TargetVelocity := [ 0.00000000000000000000, 0.00000000000000000000, 0.00000000000000000000 ],
    TargetAcceleration := [ -145.73534974155302279542, -148.36578074146780181763, 565.35337574115942516073 ]
  );
  
  positionExtrema : Struckig.PositionExtremaDesc;
END_VAR
TEST('Trajectory_HasTargetAcceleration_57');

ruckig();

// Check total duration of profiles
AssertEquals_LREAL(Expected := 0.16010935183593069664, Actual := ruckig.Duration, DELTA := 1E-8, Message := 'Duration incorrect');

// Check duration for each phase
positionExtrema := ruckig._profiles[0].positionExtrema();
AssertEquals_LREAL(0.04108196819819977946, positionExtrema.Tmax, 1E-9, message:='Profile[0] Tmax incorrect');
AssertEquals_LREAL(-33.77372971830767056645, positionExtrema.Maximum, 1E-9, message:='Profile[0] maximum incorrect');
AssertEquals_LREAL(0.00000000000000000000, positionExtrema.Tmin, 1E-9, message:='Profile[0] Tmin incorrect');
AssertEquals_LREAL(-41.78580401739355920654, positionExtrema.Minimum, 1E-9, message:='Profile[0] minimum incorrect');

positionExtrema := ruckig._profiles[1].positionExtrema();
AssertEquals_LREAL(0.16010935183593069664, positionExtrema.Tmax, 1E-9, message:='Profile[1] Tmax incorrect');
AssertEquals_LREAL(76.85926955676279703766, positionExtrema.Maximum, 1E-9, message:='Profile[1] maximum incorrect');
AssertEquals_LREAL(0.00000000000000000000, positionExtrema.Tmin, 1E-9, message:='Profile[1] Tmin incorrect');
AssertEquals_LREAL(-54.54341916085618890975, positionExtrema.Minimum, 1E-9, message:='Profile[1] minimum incorrect');

positionExtrema := ruckig._profiles[2].positionExtrema();
AssertEquals_LREAL(0.03210937502877184851, positionExtrema.Tmax, 1E-9, message:='Profile[2] Tmax incorrect');
AssertEquals_LREAL(7.08882541134368349134, positionExtrema.Maximum, 1E-9, message:='Profile[2] maximum incorrect');
AssertEquals_LREAL(0.16010935183593069664, positionExtrema.Tmin, 1E-9, message:='Profile[2] Tmin incorrect');
AssertEquals_LREAL(-20.12684108733012067205, positionExtrema.Minimum, 1E-9, message:='Profile[2] minimum incorrect');
   

TEST_FINISHED();
END_METHOD

METHOD Test_Trajectory_HasTargetAcceleration_58
VAR_INST
  ruckig : Struckig.Otg(0.001, 3) := (
  
